// TIA Portal V19 program export: 0 tag tables, 0 data types, 1 data blocks, 22 code blocks (in call order from the OBs), 0 instance data blocks

DATA_BLOCK "DEV_7"   // DB5
{ S7_Optimized_Access := 'TRUE' }
// stored: MemoryReserve 0
   VAR
      Convoyer : "ModuleConvoyer";
   END_VAR
   VAR RETAIN
      Retains : Struct
         ConvoyerA : Struct
            ProducedUnits : DInt;
            "Type" : SInt;
         END_STRUCT;
         ConvoyerB : Struct
            ProducedUnits : DInt;
            "Type" : SInt;
         END_STRUCT;
      END_STRUCT;
      Recipes : Struct
         Convoyer : Struct
            "A" : Struct
               "Type" : SInt;
               StampingPL : Struct
                  Enable : Bool := TRUE;
                  Double : Bool;
                  SecondPush : Bool;
                  SecondPreasure : Real;
                  RegularPreasure : Real := 1.3;
                  MaxPreasure : Real := 4.0;
                  TimerMaxPreasure : Time := T#1300ms;
                  TimerStamping : Time := T#400ms;
                  TimerSecond : Time;
               END_STRUCT;
               SettingsPL : Struct
                  Camera : Bool := TRUE;
                  Blow : Bool := TRUE;
                  BlowTime : Time := T#1000ms;
               END_STRUCT;
               StampingCN : Struct
                  Enable : Bool := TRUE;
                  Double : Bool;
                  SecondPush : Bool := TRUE;
                  SecondPreasure : Real := 4.0;
                  RegularPreasure : Real := 1.3;
                  MaxPreasure : Real := 4.5;
                  TimerMaxPreasure : Time := T#1300ms;
                  TimerStamping : Time := T#800ms;
                  TimerSecond : Time := T#500ms;
               END_STRUCT;
               SettingsCN : Struct
                  Camera : Bool := TRUE;
                  Blow : Bool := TRUE;
                  BlowTime : Time := T#1000ms;
               END_STRUCT;
               StampingPlastic : Struct
                  Enable : Bool := TRUE;
                  Double : Bool;
                  SecondPush : Bool;
                  SecondPreasure : Real;
                  RegularPreasure : Real := 1.3;
                  MaxPreasure : Real := 4.0;
                  TimerMaxPreasure : Time := T#1300ms;
                  TimerStamping : Time := T#400ms;
                  TimerSecond : Time;
               END_STRUCT;
               SettingsPlastic : Struct
                  Camera : Bool := TRUE;
                  Blow : Bool := TRUE;
                  BlowTime : Time := T#1000ms;
               END_STRUCT;
               StampingTransport : Struct
                  Enable : Bool := FALSE;
                  Double : Bool := FALSE;
                  SecondPush : Bool := FALSE;
                  SecondPreasure : Real;
                  RegularPreasure : Real := 1.3;
                  MaxPreasure : Real := 4.0;
                  TimerMaxPreasure : Time := T#1300ms;
                  TimerStamping : Time := T#400ms;
                  TimerSecond : Time;
               END_STRUCT;
               SettingsTransport : Struct
                  Camera : Bool := FALSE;
                  Blow : Bool := FALSE;
                  BlowTime : Time := T#1000ms;
               END_STRUCT;
            END_STRUCT;
            "B" : Struct
               "Type" : SInt;
               StampingPL : Struct
                  Enable : Bool := TRUE;
                  Double : Bool;
                  SecondPush : Bool;
                  SecondPreasure : Real;
                  RegularPreasure : Real := 1.3;
                  MaxPreasure : Real := 4.0;
                  TimerMaxPreasure : Time := T#1300ms;
                  TimerStamping : Time := T#400ms;
                  TimerSecond : Time;
               END_STRUCT;
               SettingsPL : Struct
                  Camera : Bool := TRUE;
                  Blow : Bool := TRUE;
                  BlowTime : Time := T#1000ms;
               END_STRUCT;
               StampingCN : Struct
                  Enable : Bool := TRUE;
                  Double : Bool;
                  SecondPush : Bool := TRUE;
                  SecondPreasure : Real := 4.0;
                  RegularPreasure : Real := 1.3;
                  MaxPreasure : Real := 4.5;
                  TimerMaxPreasure : Time := T#1300ms;
                  TimerStamping : Time := T#800ms;
                  TimerSecond : Time := T#500ms;
               END_STRUCT;
               SettingsCN : Struct
                  Camera : Bool := TRUE;
                  Blow : Bool := TRUE;
                  BlowTime : Time := T#1000ms;
               END_STRUCT;
               StampingPlastic : Struct
                  Enable : Bool := TRUE;
                  Double : Bool;
                  SecondPush : Bool;
                  SecondPreasure : Real;
                  RegularPreasure : Real := 1.3;
                  MaxPreasure : Real := 4.0;
                  TimerMaxPreasure : Time := T#1300ms;
                  TimerStamping : Time := T#400ms;
                  TimerSecond : Time;
               END_STRUCT;
               SettingsPlastic : Struct
                  Camera : Bool := TRUE;
                  Blow : Bool := TRUE;
                  BlowTime : Time := T#1000ms;
               END_STRUCT;
               StampingTransport : Struct
                  Enable : Bool := FALSE;
                  Double : Bool := FALSE;
                  SecondPush : Bool := FALSE;
                  SecondPreasure : Real;
                  RegularPreasure : Real := 1.3;
                  MaxPreasure : Real := 4.0;
                  TimerMaxPreasure : Time := T#1300ms;
                  TimerStamping : Time := T#400ms;
                  TimerSecond : Time;
               END_STRUCT;
               SettingsTransport : Struct
                  Camera : Bool := FALSE;
                  Blow : Bool := FALSE;
                  BlowTime : Time := T#1000ms;
               END_STRUCT;
            END_STRUCT;
         END_STRUCT;
      END_STRUCT;
      OPC : Struct
         Convoyer : Struct
            "A" : Struct
               LifetimeProduction : DInt;
               CycleTime : Time;
               CameraCycle : Time;
               StampingCycle : Time;
               ActualRecipe : WString[30];
               Status : Struct
                  ReadyToWork : Bool;
                  Working : Bool;
                  Error : Bool;
               END_STRUCT;
            END_STRUCT;
            "B" : Struct
               LifetimeProduction : DInt;
               CycleTime : Time;
               CameraCycle : Time;
               StampingCycle : Time;
               ActualRecipe : WString[30];
               Status : Struct
                  ReadyToWork : Bool;
                  Working : Bool;
                  Error : Bool;
               END_STRUCT;
            END_STRUCT;
         END_STRUCT;
      END_STRUCT;
   END_VAR
BEGIN
   Convoyer.Modular_A.CameraConnection.InterfaceId := 64;
   Convoyer.Modular_A.CameraConnection.ID := 1;
   Convoyer.Modular_A.CameraConnection.ConnectionType := 16#0B;
   Convoyer.Modular_A.CameraConnection.ActiveEstablished := false;
   Convoyer.Modular_A.CameraConnection.RemoteAddress.ADDR[1] := 192;
   Convoyer.Modular_A.CameraConnection.RemoteAddress.ADDR[2] := 168;
   Convoyer.Modular_A.CameraConnection.RemoteAddress.ADDR[3] := 0;
   Convoyer.Modular_A.CameraConnection.RemoteAddress.ADDR[4] := 70;
   Convoyer.Modular_A.CameraConnection.RemotePort := 0;
   Convoyer.Modular_A.CameraConnection.LocalPort := 2137;
   Convoyer.Modular_A.Pneumatics.Stamping.Timers.In := T#6000ms;
   Convoyer.Modular_A.Pneumatics.Stamping.Timers.Out := T#5000ms;
   Convoyer.Modular_A.Pneumatics.IVT.Sensor.Analog.SetValue := 0.0;
   Convoyer.Modular_A.Pneumatics.IVT.Sensor.Settings.Min := 0.0;
   Convoyer.Modular_A.Pneumatics.IVT.Sensor.Settings.Max := 7.0;
   Convoyer.Modular_A.HMI.Camera.Enable := TRUE;
   Convoyer.Modular_A.HMI.Camera.TimerConnection := T#100000ms;
   Convoyer.Modular_A.HMI.Stamping.Enable := TRUE;
   Convoyer.Modular_A.HMI.Stamping.RegularPreasure := 3.0;
   Convoyer.Modular_A.HMI.Stamping.MaxPreasure := 6.0;
   Convoyer.Modular_A.HMI.Stamping.TimerMaxPreasure := T#1500ms;
   Convoyer.Modular_A.HMI.Stamping.TimerStamping := T#1000ms;
   Convoyer.Modular_A.HMI.Blow.Enable := TRUE;
   Convoyer.Modular_A.HMI.Blow."Time" := T#1000ms;
   Convoyer.Modular_B.CameraConnection.InterfaceId := 64;
   Convoyer.Modular_B.CameraConnection.ID := 16#2;
   Convoyer.Modular_B.CameraConnection.ConnectionType := 16#0B;
   Convoyer.Modular_B.CameraConnection.ActiveEstablished := FALSE;
   Convoyer.Modular_B.CameraConnection.RemoteAddress.ADDR[1] := 192;
   Convoyer.Modular_B.CameraConnection.RemoteAddress.ADDR[2] := 168;
   Convoyer.Modular_B.CameraConnection.RemoteAddress.ADDR[3] := 0;
   Convoyer.Modular_B.CameraConnection.RemoteAddress.ADDR[4] := 71;
   Convoyer.Modular_B.CameraConnection.RemotePort := 0;
   Convoyer.Modular_B.CameraConnection.LocalPort := 2137;
END_DATA_BLOCK

ORGANIZATION_BLOCK "Main"   // OB1, LAD, ProgramCycle
TITLE = "Main Program Sweep (Cycle)"
{ S7_Optimized_Access := 'TRUE' }
// stored: SetENOAutomatically false
   VAR_INPUT
      Initial_Call : Bool;   // Initial call of this OB
      Remanence : Bool;   // =True, if remanent data are available
   END_VAR
BEGIN

REGION Network 1
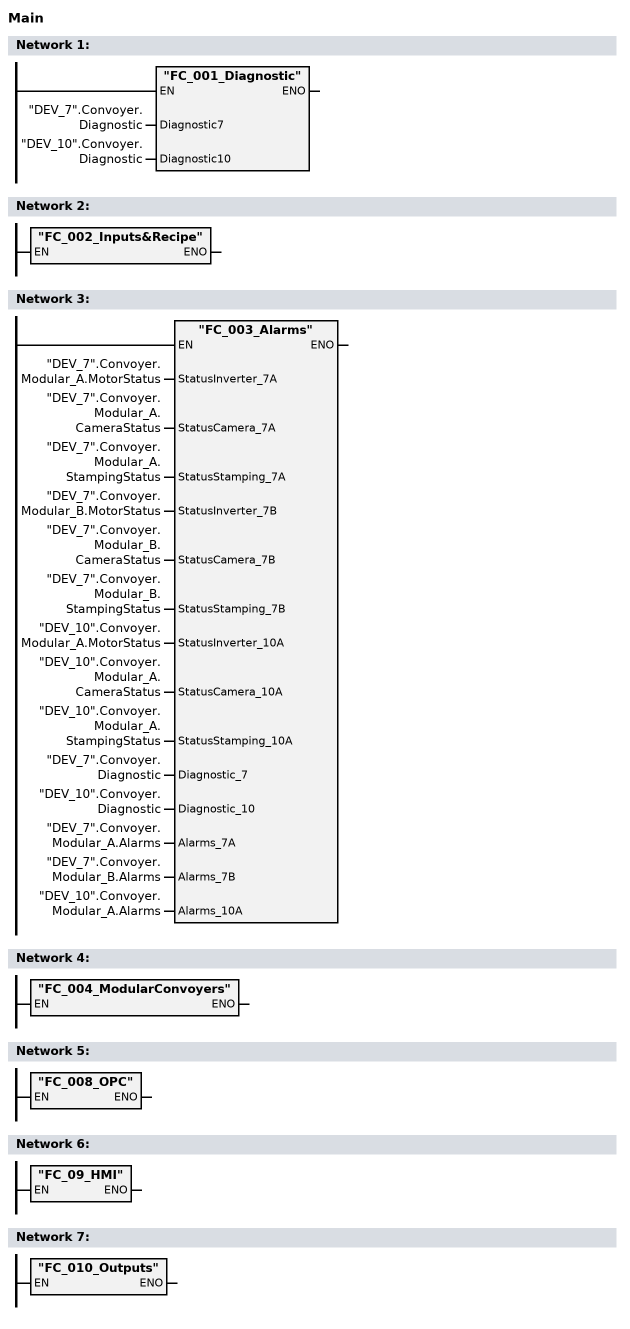
   RUNG wire#powerrail
      "FC_001_Diagnostic"(Diagnostic7 := "DEV_7".Convoyer.Diagnostic, Diagnostic10 := "DEV_10".Convoyer.Diagnostic)
   END_RUNG
   // the same network as SCL:
   "FC_001_Diagnostic"(Diagnostic7 := "DEV_7".Convoyer.Diagnostic, Diagnostic10 := "DEV_10".Convoyer.Diagnostic);
END_REGION

REGION Network 2
   RUNG wire#powerrail
      "FC_002_Inputs&Recipe"()
   END_RUNG
   // the same network as SCL:
   "FC_002_Inputs&Recipe"();
END_REGION

REGION Network 3
   RUNG wire#powerrail
      "FC_003_Alarms"(StatusInverter_7A := "DEV_7".Convoyer.Modular_A.MotorStatus, StatusCamera_7A := "DEV_7".Convoyer.Modular_A.CameraStatus, StatusStamping_7A := "DEV_7".Convoyer.Modular_A.StampingStatus, StatusInverter_7B := "DEV_7".Convoyer.Modular_B.MotorStatus, StatusCamera_7B := "DEV_7".Convoyer.Modular_B.CameraStatus, StatusStamping_7B := "DEV_7".Convoyer.Modular_B.StampingStatus, StatusInverter_10A := "DEV_10".Convoyer.Modular_A.MotorStatus, StatusCamera_10A := "DEV_10".Convoyer.Modular_A.CameraStatus, StatusStamping_10A := "DEV_10".Convoyer.Modular_A.StampingStatus, Diagnostic_7 := "DEV_7".Convoyer.Diagnostic, Diagnostic_10 := "DEV_10".Convoyer.Diagnostic, Alarms_7A := "DEV_7".Convoyer.Modular_A.Alarms, Alarms_7B := "DEV_7".Convoyer.Modular_B.Alarms, Alarms_10A := "DEV_10".Convoyer.Modular_A.Alarms)
   END_RUNG
   // the same network as SCL:
   "FC_003_Alarms"(StatusInverter_7A := "DEV_7".Convoyer.Modular_A.MotorStatus,
                   StatusCamera_7A := "DEV_7".Convoyer.Modular_A.CameraStatus,
                   StatusStamping_7A := "DEV_7".Convoyer.Modular_A.StampingStatus,
                   StatusInverter_7B := "DEV_7".Convoyer.Modular_B.MotorStatus,
                   StatusCamera_7B := "DEV_7".Convoyer.Modular_B.CameraStatus,
                   StatusStamping_7B := "DEV_7".Convoyer.Modular_B.StampingStatus,
                   StatusInverter_10A := "DEV_10".Convoyer.Modular_A.MotorStatus,
                   StatusCamera_10A := "DEV_10".Convoyer.Modular_A.CameraStatus,
                   StatusStamping_10A := "DEV_10".Convoyer.Modular_A.StampingStatus,
                   Diagnostic_7 := "DEV_7".Convoyer.Diagnostic,
                   Diagnostic_10 := "DEV_10".Convoyer.Diagnostic,
                   Alarms_7A := "DEV_7".Convoyer.Modular_A.Alarms,
                   Alarms_7B := "DEV_7".Convoyer.Modular_B.Alarms,
                   Alarms_10A := "DEV_10".Convoyer.Modular_A.Alarms);
END_REGION

REGION Network 4
   RUNG wire#powerrail
      "FC_004_ModularConvoyers"()
   END_RUNG
   // the same network as SCL:
   "FC_004_ModularConvoyers"();
END_REGION

REGION Network 5
   RUNG wire#powerrail
      "FC_008_OPC"()
   END_RUNG
   // the same network as SCL:
   "FC_008_OPC"();
END_REGION

REGION Network 6
   RUNG wire#powerrail
      "FC_09_HMI"()
   END_RUNG
   // the same network as SCL:
   "FC_09_HMI"();
END_REGION

REGION Network 7
   RUNG wire#powerrail
      "FC_010_Outputs"()
   END_RUNG
   // the same network as SCL:
   "FC_010_Outputs"();
END_REGION
END_ORGANIZATION_BLOCK

FUNCTION "FC_001_Diagnostic" : Void   // FC12, LAD
{ S7_Optimized_Access := 'TRUE' }
// stored: SetENOAutomatically false
   VAR_IN_OUT
      Diagnostic7 : "DiagnosticMainCabinet";
      Diagnostic10 : "DiagnosticMainCabinet";
   END_VAR
BEGIN

REGION Network 1 (SCL)
   //************************************************************
   //===Author: Mateusz Połojko
   //-----Linkedin: https://pl.linkedin.com/in/mateusz-po%C5%82ojko-52a3541b1
   //-----Github: https://github.com/Bhazel95
   //===Description:
   //-----Diagnostic of hardware components
   //===Customer:
   //-----Apator Powogaz S.A.
   //************************************************************
END_REGION

REGION Network 2 (SCL)
   //Transporter 7A & 7B
   #Diagnostic7.ET_200SP.HeadModule_0.LADDR:= "IO_device_1~Head";
   #Diagnostic7.ET_200SP.HeadModule_0.Mode := 1;

   #Diagnostic7.ET_200SP.BusAdapter_1.LADDR := "IO_device_1~BusAdapter-Send_1xFC_1";
   #Diagnostic7.ET_200SP.BusAdapter_1.Mode := 1;

   #Diagnostic7.ET_200SP.InputSafety_2.LADDR := "IO_device_1~F-DI_8x24VDC_HF_1" ;
   #Diagnostic7.ET_200SP.InputSafety_2.Mode := 1;

   #Diagnostic7.ET_200SP.InputSafety_3.LADDR := "IO_device_1~F-DI_8x24VDC_HF_2";
   #Diagnostic7.ET_200SP.InputSafety_3.Mode := 1;

   #Diagnostic7.ET_200SP.InputSafety_4.LADDR := "IO_device_1~F-DI_8x24VDC_HF_3";
   #Diagnostic7.ET_200SP.InputSafety_4.Mode := 1;

   #Diagnostic7.ET_200SP.InputSafety_5.LADDR := "IO_device_1~F-DI_8x24VDC_HF_5";
   #Diagnostic7.ET_200SP.InputSafety_5.Mode := 1;

   #Diagnostic7.ET_200SP.InputSafety_6.LADDR := "IO_device_1~F-DI_8x24VDC_HF_4";
   #Diagnostic7.ET_200SP.InputSafety_6.Mode := 1;

   #Diagnostic7.ET_200SP.OutputSafety_7.LADDR := "IO_device_1~F-DQ_8x24VDC_0_5A_PP_HF_1";
   #Diagnostic7.ET_200SP.OutputSafety_7.Mode := 1;

   #Diagnostic7.ET_200SP.RelaySafety_9.LADDR := "IO_device_1~F-RQ_1x24__48VDC_24__230VAC_5A_1";
   #Diagnostic7.ET_200SP.RelaySafety_9.Mode := 1;

   #Diagnostic7.ET_200SP.RelaySafety_10.LADDR := "IO_device_1~F-RQ_1x24__48VDC_24__230VAC_5A_2";
   #Diagnostic7.ET_200SP.RelaySafety_10.Mode := 1;

   #Diagnostic7.ET_200SP.InputsDigital_11.LADDR := "IO_device_1~DI_16x24VDC_ST_1";
   #Diagnostic7.ET_200SP.InputsDigital_11.Mode := 1;

   #Diagnostic7.ET_200SP.InputsDigital_12.LADDR := "IO_device_1~DI_16x24VDC_ST_2";
   #Diagnostic7.ET_200SP.InputsDigital_12.Mode := 1;

   #Diagnostic7.ET_200SP.InputsDigital_13.LADDR := "IO_device_1~DI_16x24VDC_ST_3";
   #Diagnostic7.ET_200SP.InputsDigital_13.Mode := 1;

   #Diagnostic7.ET_200SP.InputAnalog_14.LADDR := "IO_device_1~AI_2xI_2-_4-wire_ST_1";
   #Diagnostic7.ET_200SP.InputAnalog_14.Mode := 1;

   #Diagnostic7.ET_200SP.OutputDigital_15.LADDR := "IO_device_1~DQ_16x24VDC_0_5A_ST_1";
   #Diagnostic7.ET_200SP.OutputDigital_15.Mode := 1;

   #Diagnostic7.ET_200SP.OutputDigital_16.LADDR := "IO_device_1~DQ_16x24VDC_0_5A_ST_2";
   #Diagnostic7.ET_200SP.OutputDigital_16.Mode := 1;

   #Diagnostic7.ET_200SP.OutputDigital_17.LADDR := "IO_device_1~DQ_16x24VDC_0_5A_ST_3";
   #Diagnostic7.ET_200SP.OutputDigital_17.Mode := 1;

   #Diagnostic7.ET_200SP.OutputDigital_18.LADDR := "IO_device_1~DQ_16x24VDC_0_5A_ST_4";
   #Diagnostic7.ET_200SP.OutputDigital_18.Mode := 1;

   #Diagnostic7.ET_200SP.OutputAnalog_19.LADDR := "IO_device_1~AQ_2xI_ST_1";
   #Diagnostic7.ET_200SP.OutputAnalog_19.Mode := 1;

   #Diagnostic7.ET_200SP.ET_200AL_1.LADDR := "IO_device_1~DI_8x24VDC_8xM8_1";
   #Diagnostic7.ET_200SP.ET_200AL_1.Mode := 1;

   #Diagnostic7.ET_200SP.ET_200AL_2.LADDR := "IO_device_1~DI_8x24VDC_8xM8_2";
   #Diagnostic7.ET_200SP.ET_200AL_2.Mode := 1;


   #Diagnostic7.SinamicG120_1.LADDR := "G120_CU250S_2_PN_VECTOR_7A~PROFINET_interface~IODevice";
   #Diagnostic7.SinamicG120_1.Mode := 1;

   #Diagnostic7.SinamicG120_1.LADDR := "G120_CU250S_2_PN_VECTOR_7B~PROFINET_interface~IODevice";
   #Diagnostic7.SinamicG120_1.Mode := 1;
END_REGION

REGION Network 3 (SCL)
   //Transporter 10A & 10B
   #Diagnostic10.ET_200SP.HeadModule_0.LADDR := "IO_device_2~Head";
   #Diagnostic10.ET_200SP.HeadModule_0.Mode := 1;

   #Diagnostic10.ET_200SP.BusAdapter_1.LADDR := "IO_device_2~BusAdapter-Send_1xFC_1";
   #Diagnostic10.ET_200SP.BusAdapter_1.Mode := 1;

   #Diagnostic10.ET_200SP.InputSafety_2.LADDR := "IO_device_2~F-DI_8x24VDC_HF_1";
   #Diagnostic10.ET_200SP.InputSafety_2.Mode := 1;

   #Diagnostic10.ET_200SP.InputSafety_3.LADDR := "IO_device_2~F-DI_8x24VDC_HF_2";
   #Diagnostic10.ET_200SP.InputSafety_3.Mode := 1;

   #Diagnostic10.ET_200SP.InputSafety_4.LADDR := "IO_device_2~F-DI_8x24VDC_HF_3";
   #Diagnostic10.ET_200SP.InputSafety_4.Mode := 1;

   #Diagnostic10.ET_200SP.InputSafety_5.LADDR := "IO_device_2~F-DI_8x24VDC_HF_4";
   #Diagnostic10.ET_200SP.InputSafety_5.Mode := 1;

   #Diagnostic10.ET_200SP.InputSafety_6.LADDR := "IO_device_2~F-DI_8x24VDC_HF_5";
   #Diagnostic10.ET_200SP.InputSafety_6.Mode := 1;

   #Diagnostic10.ET_200SP.OutputSafety_7.LADDR := "IO_device_2~F-DQ_8x24VDC_0_5A_PP_HF_1";
   #Diagnostic10.ET_200SP.OutputSafety_7.Mode := 1;

   #Diagnostic10.ET_200SP.RelaySafety_9.LADDR := "IO_device_2~F-RQ_1x24__48VDC_24__230VAC_5A_1";
   #Diagnostic10.ET_200SP.RelaySafety_9.Mode := 1;

   #Diagnostic10.ET_200SP.RelaySafety_10.LADDR := "IO_device_2~F-RQ_1x24__48VDC_24__230VAC_5A_2";
   #Diagnostic10.ET_200SP.RelaySafety_10.Mode := 1;

   #Diagnostic10.ET_200SP.InputsDigital_11.LADDR := "IO_device_2~DI_16x24VDC_ST_1";
   #Diagnostic10.ET_200SP.InputsDigital_11.Mode := 1;

   #Diagnostic10.ET_200SP.InputsDigital_12.LADDR := "IO_device_2~DI_16x24VDC_ST_2";
   #Diagnostic10.ET_200SP.InputsDigital_12.Mode := 1;

   #Diagnostic10.ET_200SP.InputsDigital_13.LADDR := "IO_device_2~DI_16x24VDC_ST_3";
   #Diagnostic10.ET_200SP.InputsDigital_13.Mode := 1;

   #Diagnostic10.ET_200SP.InputAnalog_14.LADDR := "IO_device_2~AI_2xI_2-_4-wire_ST_1";
   #Diagnostic10.ET_200SP.InputAnalog_14.Mode := 1;

   #Diagnostic10.ET_200SP.OutputDigital_15.LADDR := "IO_device_2~DQ_16x24VDC_0_5A_ST_1";
   #Diagnostic10.ET_200SP.OutputDigital_15.Mode := 1;

   #Diagnostic10.ET_200SP.OutputDigital_16.LADDR := "IO_device_2~DQ_16x24VDC_0_5A_ST_2";
   #Diagnostic10.ET_200SP.OutputDigital_16.Mode := 1;

   #Diagnostic10.ET_200SP.OutputDigital_17.LADDR := "IO_device_2~DQ_16x24VDC_0_5A_ST_3";
   #Diagnostic10.ET_200SP.OutputDigital_17.Mode := 1;

   #Diagnostic10.ET_200SP.OutputDigital_18.LADDR := "IO_device_2~DQ_16x24VDC_0_5A_ST_4";
   #Diagnostic10.ET_200SP.OutputDigital_18.Mode := 1;

   #Diagnostic10.ET_200SP.OutputAnalog_19.LADDR := "IO_device_2~AQ_2xI_ST_1";
   #Diagnostic10.ET_200SP.OutputAnalog_19.Mode := 1;

   #Diagnostic10.ET_200SP.ET_200AL_1.LADDR := "IO_device_2~DI_8x24VDC_8xM8_1";
   #Diagnostic10.ET_200SP.ET_200AL_1.Mode := 1;

   #Diagnostic10.ET_200SP.ET_200AL_2.LADDR := "IO_device_2~DI_8x24VDC_8xM8_2";
   #Diagnostic10.ET_200SP.ET_200AL_2.Mode := 1;


   #Diagnostic10.SinamicG120_1.LADDR := "G120_CU250S_2_PN_VECTOR_10A~PROFINET_interface~IODevice";
   #Diagnostic10.SinamicG120_1.Mode := 1;
END_REGION

REGION Network 4
   // ET 200SP - MODUL GLOWNY 7
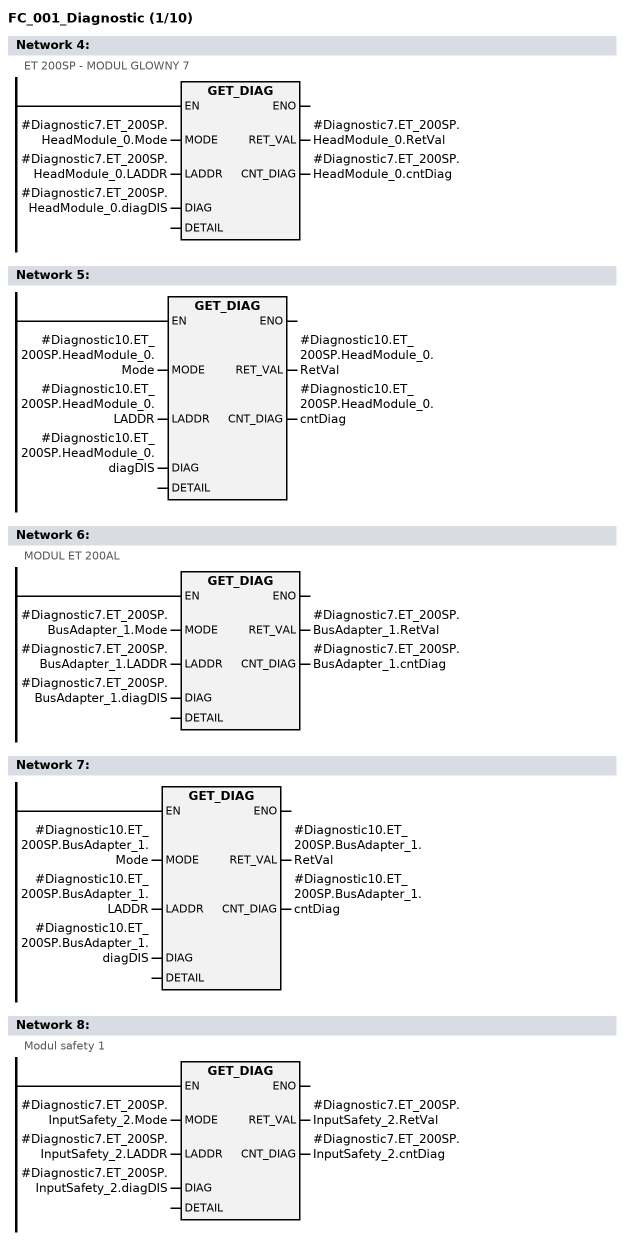
   RUNG wire#powerrail
      GET_DIAG(MODE := #Diagnostic7.ET_200SP.HeadModule_0.Mode, LADDR := #Diagnostic7.ET_200SP.HeadModule_0.LADDR, DIAG := #Diagnostic7.ET_200SP.HeadModule_0.diagDIS, DETAIL :=, RET_VAL => #Diagnostic7.ET_200SP.HeadModule_0.RetVal, CNT_DIAG => #Diagnostic7.ET_200SP.HeadModule_0.cntDiag)
   END_RUNG
   // the same network as SCL:
   #Diagnostic7.ET_200SP.HeadModule_0.RetVal := GET_DIAG(MODE := #Diagnostic7.ET_200SP.HeadModule_0.Mode,
                           LADDR := #Diagnostic7.ET_200SP.HeadModule_0.LADDR,
                           DIAG := #Diagnostic7.ET_200SP.HeadModule_0.diagDIS,
                           CNT_DIAG => #Diagnostic7.ET_200SP.HeadModule_0.cntDiag);
END_REGION

REGION Network 5
   RUNG wire#powerrail
      GET_DIAG(MODE := #Diagnostic10.ET_200SP.HeadModule_0.Mode, LADDR := #Diagnostic10.ET_200SP.HeadModule_0.LADDR, DIAG := #Diagnostic10.ET_200SP.HeadModule_0.diagDIS, DETAIL :=, RET_VAL => #Diagnostic10.ET_200SP.HeadModule_0.RetVal, CNT_DIAG => #Diagnostic10.ET_200SP.HeadModule_0.cntDiag)
   END_RUNG
   // the same network as SCL:
   #Diagnostic10.ET_200SP.HeadModule_0.RetVal := GET_DIAG(MODE := #Diagnostic10.ET_200SP.HeadModule_0.Mode,
                           LADDR := #Diagnostic10.ET_200SP.HeadModule_0.LADDR,
                           DIAG := #Diagnostic10.ET_200SP.HeadModule_0.diagDIS,
                           CNT_DIAG => #Diagnostic10.ET_200SP.HeadModule_0.cntDiag);
END_REGION

REGION Network 6
   // MODUL ET 200AL
   RUNG wire#powerrail
      GET_DIAG(MODE := #Diagnostic7.ET_200SP.BusAdapter_1.Mode, LADDR := #Diagnostic7.ET_200SP.BusAdapter_1.LADDR, DIAG := #Diagnostic7.ET_200SP.BusAdapter_1.diagDIS, DETAIL :=, RET_VAL => #Diagnostic7.ET_200SP.BusAdapter_1.RetVal, CNT_DIAG => #Diagnostic7.ET_200SP.BusAdapter_1.cntDiag)
   END_RUNG
   // the same network as SCL:
   #Diagnostic7.ET_200SP.BusAdapter_1.RetVal := GET_DIAG(MODE := #Diagnostic7.ET_200SP.BusAdapter_1.Mode,
                           LADDR := #Diagnostic7.ET_200SP.BusAdapter_1.LADDR,
                           DIAG := #Diagnostic7.ET_200SP.BusAdapter_1.diagDIS,
                           CNT_DIAG => #Diagnostic7.ET_200SP.BusAdapter_1.cntDiag);
END_REGION

REGION Network 7
   RUNG wire#powerrail
      GET_DIAG(MODE := #Diagnostic10.ET_200SP.BusAdapter_1.Mode, LADDR := #Diagnostic10.ET_200SP.BusAdapter_1.LADDR, DIAG := #Diagnostic10.ET_200SP.BusAdapter_1.diagDIS, DETAIL :=, RET_VAL => #Diagnostic10.ET_200SP.BusAdapter_1.RetVal, CNT_DIAG => #Diagnostic10.ET_200SP.BusAdapter_1.cntDiag)
   END_RUNG
   // the same network as SCL:
   #Diagnostic10.ET_200SP.BusAdapter_1.RetVal := GET_DIAG(MODE := #Diagnostic10.ET_200SP.BusAdapter_1.Mode,
                           LADDR := #Diagnostic10.ET_200SP.BusAdapter_1.LADDR,
                           DIAG := #Diagnostic10.ET_200SP.BusAdapter_1.diagDIS,
                           CNT_DIAG => #Diagnostic10.ET_200SP.BusAdapter_1.cntDiag);
END_REGION

REGION Network 8
   // Modul safety 1
   RUNG wire#powerrail
      GET_DIAG(MODE := #Diagnostic7.ET_200SP.InputSafety_2.Mode, LADDR := #Diagnostic7.ET_200SP.InputSafety_2.LADDR, DIAG := #Diagnostic7.ET_200SP.InputSafety_2.diagDIS, DETAIL :=, RET_VAL => #Diagnostic7.ET_200SP.InputSafety_2.RetVal, CNT_DIAG => #Diagnostic7.ET_200SP.InputSafety_2.cntDiag)
   END_RUNG
   // the same network as SCL:
   #Diagnostic7.ET_200SP.InputSafety_2.RetVal := GET_DIAG(MODE := #Diagnostic7.ET_200SP.InputSafety_2.Mode,
                           LADDR := #Diagnostic7.ET_200SP.InputSafety_2.LADDR,
                           DIAG := #Diagnostic7.ET_200SP.InputSafety_2.diagDIS,
                           CNT_DIAG => #Diagnostic7.ET_200SP.InputSafety_2.cntDiag);
END_REGION

REGION Network 9
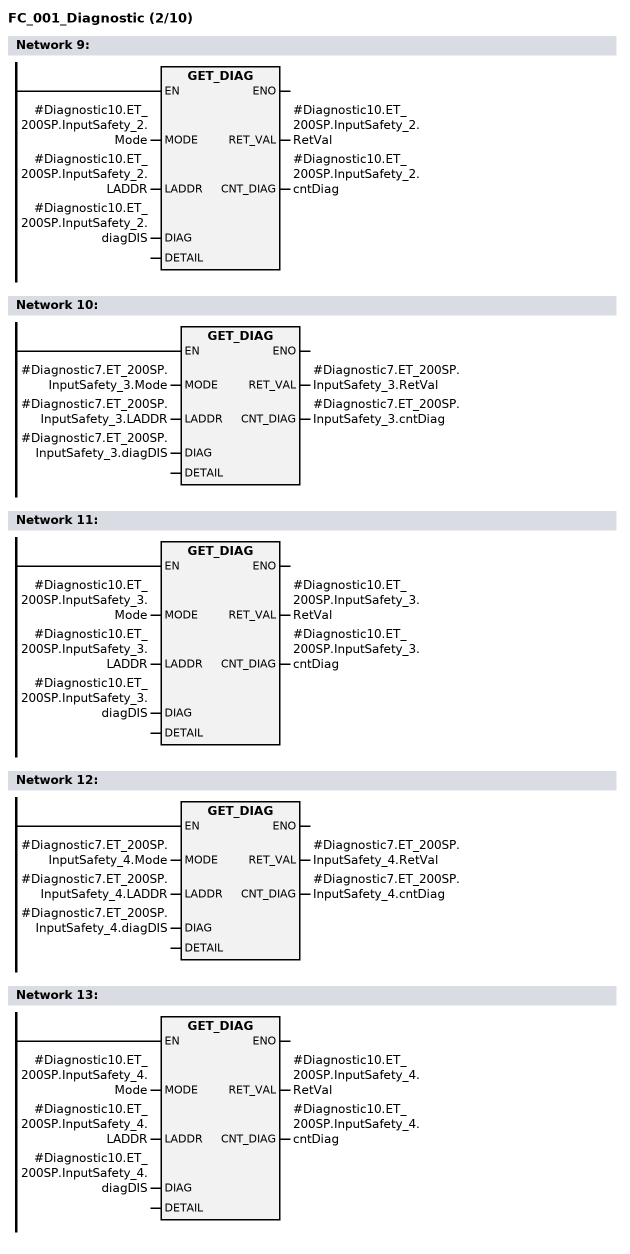
   RUNG wire#powerrail
      GET_DIAG(MODE := #Diagnostic10.ET_200SP.InputSafety_2.Mode, LADDR := #Diagnostic10.ET_200SP.InputSafety_2.LADDR, DIAG := #Diagnostic10.ET_200SP.InputSafety_2.diagDIS, DETAIL :=, RET_VAL => #Diagnostic10.ET_200SP.InputSafety_2.RetVal, CNT_DIAG => #Diagnostic10.ET_200SP.InputSafety_2.cntDiag)
   END_RUNG
   // the same network as SCL:
   #Diagnostic10.ET_200SP.InputSafety_2.RetVal := GET_DIAG(MODE := #Diagnostic10.ET_200SP.InputSafety_2.Mode,
                           LADDR := #Diagnostic10.ET_200SP.InputSafety_2.LADDR,
                           DIAG := #Diagnostic10.ET_200SP.InputSafety_2.diagDIS,
                           CNT_DIAG => #Diagnostic10.ET_200SP.InputSafety_2.cntDiag);
END_REGION

REGION Network 10
   RUNG wire#powerrail
      GET_DIAG(MODE := #Diagnostic7.ET_200SP.InputSafety_3.Mode, LADDR := #Diagnostic7.ET_200SP.InputSafety_3.LADDR, DIAG := #Diagnostic7.ET_200SP.InputSafety_3.diagDIS, DETAIL :=, RET_VAL => #Diagnostic7.ET_200SP.InputSafety_3.RetVal, CNT_DIAG => #Diagnostic7.ET_200SP.InputSafety_3.cntDiag)
   END_RUNG
   // the same network as SCL:
   #Diagnostic7.ET_200SP.InputSafety_3.RetVal := GET_DIAG(MODE := #Diagnostic7.ET_200SP.InputSafety_3.Mode,
                           LADDR := #Diagnostic7.ET_200SP.InputSafety_3.LADDR,
                           DIAG := #Diagnostic7.ET_200SP.InputSafety_3.diagDIS,
                           CNT_DIAG => #Diagnostic7.ET_200SP.InputSafety_3.cntDiag);
END_REGION

REGION Network 11
   RUNG wire#powerrail
      GET_DIAG(MODE := #Diagnostic10.ET_200SP.InputSafety_3.Mode, LADDR := #Diagnostic10.ET_200SP.InputSafety_3.LADDR, DIAG := #Diagnostic10.ET_200SP.InputSafety_3.diagDIS, DETAIL :=, RET_VAL => #Diagnostic10.ET_200SP.InputSafety_3.RetVal, CNT_DIAG => #Diagnostic10.ET_200SP.InputSafety_3.cntDiag)
   END_RUNG
   // the same network as SCL:
   #Diagnostic10.ET_200SP.InputSafety_3.RetVal := GET_DIAG(MODE := #Diagnostic10.ET_200SP.InputSafety_3.Mode,
                           LADDR := #Diagnostic10.ET_200SP.InputSafety_3.LADDR,
                           DIAG := #Diagnostic10.ET_200SP.InputSafety_3.diagDIS,
                           CNT_DIAG => #Diagnostic10.ET_200SP.InputSafety_3.cntDiag);
END_REGION

REGION Network 12
   RUNG wire#powerrail
      GET_DIAG(MODE := #Diagnostic7.ET_200SP.InputSafety_4.Mode, LADDR := #Diagnostic7.ET_200SP.InputSafety_4.LADDR, DIAG := #Diagnostic7.ET_200SP.InputSafety_4.diagDIS, DETAIL :=, RET_VAL => #Diagnostic7.ET_200SP.InputSafety_4.RetVal, CNT_DIAG => #Diagnostic7.ET_200SP.InputSafety_4.cntDiag)
   END_RUNG
   // the same network as SCL:
   #Diagnostic7.ET_200SP.InputSafety_4.RetVal := GET_DIAG(MODE := #Diagnostic7.ET_200SP.InputSafety_4.Mode,
                           LADDR := #Diagnostic7.ET_200SP.InputSafety_4.LADDR,
                           DIAG := #Diagnostic7.ET_200SP.InputSafety_4.diagDIS,
                           CNT_DIAG => #Diagnostic7.ET_200SP.InputSafety_4.cntDiag);
END_REGION

REGION Network 13
   RUNG wire#powerrail
      GET_DIAG(MODE := #Diagnostic10.ET_200SP.InputSafety_4.Mode, LADDR := #Diagnostic10.ET_200SP.InputSafety_4.LADDR, DIAG := #Diagnostic10.ET_200SP.InputSafety_4.diagDIS, DETAIL :=, RET_VAL => #Diagnostic10.ET_200SP.InputSafety_4.RetVal, CNT_DIAG => #Diagnostic10.ET_200SP.InputSafety_4.cntDiag)
   END_RUNG
   // the same network as SCL:
   #Diagnostic10.ET_200SP.InputSafety_4.RetVal := GET_DIAG(MODE := #Diagnostic10.ET_200SP.InputSafety_4.Mode,
                           LADDR := #Diagnostic10.ET_200SP.InputSafety_4.LADDR,
                           DIAG := #Diagnostic10.ET_200SP.InputSafety_4.diagDIS,
                           CNT_DIAG => #Diagnostic10.ET_200SP.InputSafety_4.cntDiag);
END_REGION

REGION Network 14
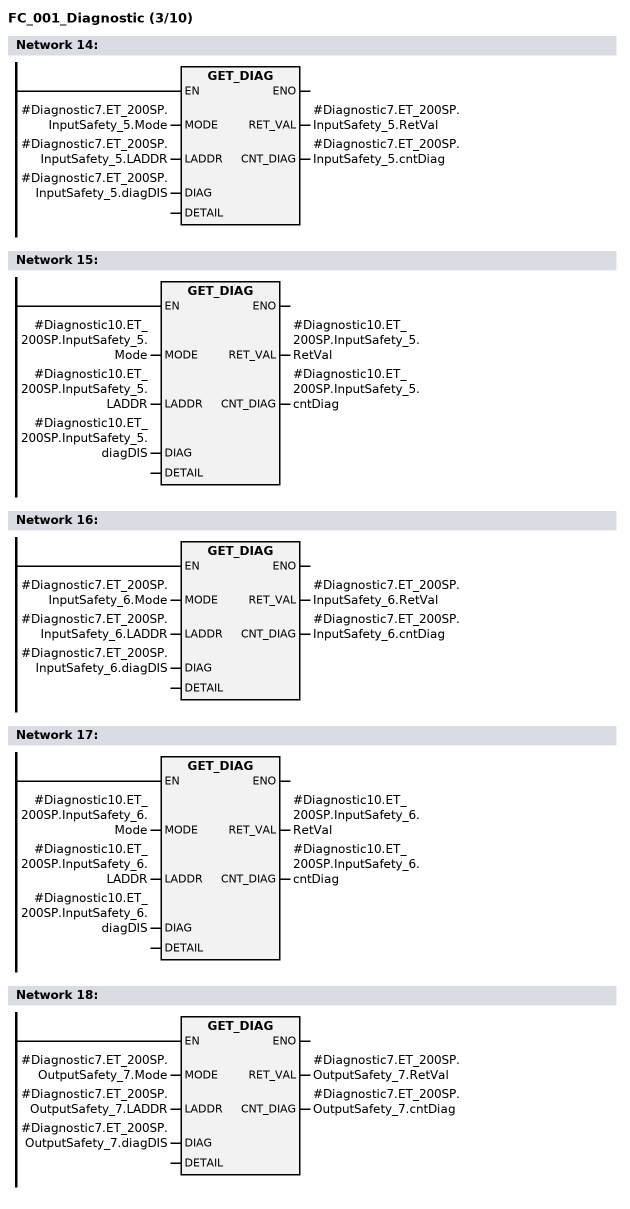
   RUNG wire#powerrail
      GET_DIAG(MODE := #Diagnostic7.ET_200SP.InputSafety_5.Mode, LADDR := #Diagnostic7.ET_200SP.InputSafety_5.LADDR, DIAG := #Diagnostic7.ET_200SP.InputSafety_5.diagDIS, DETAIL :=, RET_VAL => #Diagnostic7.ET_200SP.InputSafety_5.RetVal, CNT_DIAG => #Diagnostic7.ET_200SP.InputSafety_5.cntDiag)
   END_RUNG
   // the same network as SCL:
   #Diagnostic7.ET_200SP.InputSafety_5.RetVal := GET_DIAG(MODE := #Diagnostic7.ET_200SP.InputSafety_5.Mode,
                           LADDR := #Diagnostic7.ET_200SP.InputSafety_5.LADDR,
                           DIAG := #Diagnostic7.ET_200SP.InputSafety_5.diagDIS,
                           CNT_DIAG => #Diagnostic7.ET_200SP.InputSafety_5.cntDiag);
END_REGION

REGION Network 15
   RUNG wire#powerrail
      GET_DIAG(MODE := #Diagnostic10.ET_200SP.InputSafety_5.Mode, LADDR := #Diagnostic10.ET_200SP.InputSafety_5.LADDR, DIAG := #Diagnostic10.ET_200SP.InputSafety_5.diagDIS, DETAIL :=, RET_VAL => #Diagnostic10.ET_200SP.InputSafety_5.RetVal, CNT_DIAG => #Diagnostic10.ET_200SP.InputSafety_5.cntDiag)
   END_RUNG
   // the same network as SCL:
   #Diagnostic10.ET_200SP.InputSafety_5.RetVal := GET_DIAG(MODE := #Diagnostic10.ET_200SP.InputSafety_5.Mode,
                           LADDR := #Diagnostic10.ET_200SP.InputSafety_5.LADDR,
                           DIAG := #Diagnostic10.ET_200SP.InputSafety_5.diagDIS,
                           CNT_DIAG => #Diagnostic10.ET_200SP.InputSafety_5.cntDiag);
END_REGION

REGION Network 16
   RUNG wire#powerrail
      GET_DIAG(MODE := #Diagnostic7.ET_200SP.InputSafety_6.Mode, LADDR := #Diagnostic7.ET_200SP.InputSafety_6.LADDR, DIAG := #Diagnostic7.ET_200SP.InputSafety_6.diagDIS, DETAIL :=, RET_VAL => #Diagnostic7.ET_200SP.InputSafety_6.RetVal, CNT_DIAG => #Diagnostic7.ET_200SP.InputSafety_6.cntDiag)
   END_RUNG
   // the same network as SCL:
   #Diagnostic7.ET_200SP.InputSafety_6.RetVal := GET_DIAG(MODE := #Diagnostic7.ET_200SP.InputSafety_6.Mode,
                           LADDR := #Diagnostic7.ET_200SP.InputSafety_6.LADDR,
                           DIAG := #Diagnostic7.ET_200SP.InputSafety_6.diagDIS,
                           CNT_DIAG => #Diagnostic7.ET_200SP.InputSafety_6.cntDiag);
END_REGION

REGION Network 17
   RUNG wire#powerrail
      GET_DIAG(MODE := #Diagnostic10.ET_200SP.InputSafety_6.Mode, LADDR := #Diagnostic10.ET_200SP.InputSafety_6.LADDR, DIAG := #Diagnostic10.ET_200SP.InputSafety_6.diagDIS, DETAIL :=, RET_VAL => #Diagnostic10.ET_200SP.InputSafety_6.RetVal, CNT_DIAG => #Diagnostic10.ET_200SP.InputSafety_6.cntDiag)
   END_RUNG
   // the same network as SCL:
   #Diagnostic10.ET_200SP.InputSafety_6.RetVal := GET_DIAG(MODE := #Diagnostic10.ET_200SP.InputSafety_6.Mode,
                           LADDR := #Diagnostic10.ET_200SP.InputSafety_6.LADDR,
                           DIAG := #Diagnostic10.ET_200SP.InputSafety_6.diagDIS,
                           CNT_DIAG => #Diagnostic10.ET_200SP.InputSafety_6.cntDiag);
END_REGION

REGION Network 18
   RUNG wire#powerrail
      GET_DIAG(MODE := #Diagnostic7.ET_200SP.OutputSafety_7.Mode, LADDR := #Diagnostic7.ET_200SP.OutputSafety_7.LADDR, DIAG := #Diagnostic7.ET_200SP.OutputSafety_7.diagDIS, DETAIL :=, RET_VAL => #Diagnostic7.ET_200SP.OutputSafety_7.RetVal, CNT_DIAG => #Diagnostic7.ET_200SP.OutputSafety_7.cntDiag)
   END_RUNG
   // the same network as SCL:
   #Diagnostic7.ET_200SP.OutputSafety_7.RetVal := GET_DIAG(MODE := #Diagnostic7.ET_200SP.OutputSafety_7.Mode,
                           LADDR := #Diagnostic7.ET_200SP.OutputSafety_7.LADDR,
                           DIAG := #Diagnostic7.ET_200SP.OutputSafety_7.diagDIS,
                           CNT_DIAG => #Diagnostic7.ET_200SP.OutputSafety_7.cntDiag);
END_REGION

REGION Network 19
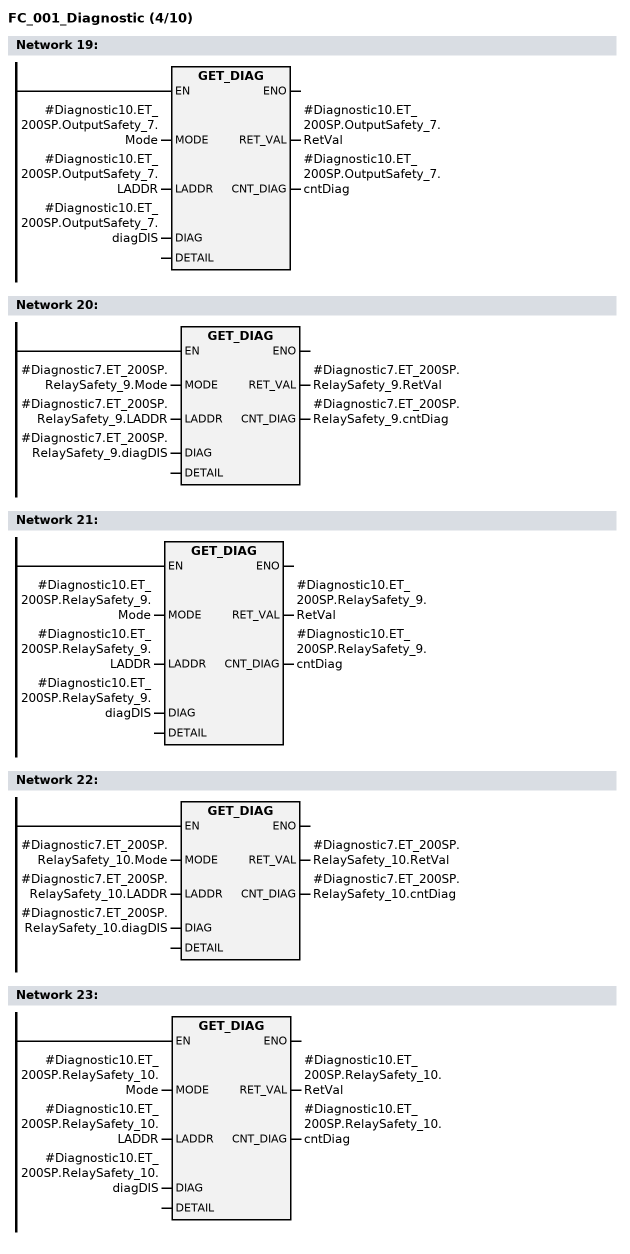
   RUNG wire#powerrail
      GET_DIAG(MODE := #Diagnostic10.ET_200SP.OutputSafety_7.Mode, LADDR := #Diagnostic10.ET_200SP.OutputSafety_7.LADDR, DIAG := #Diagnostic10.ET_200SP.OutputSafety_7.diagDIS, DETAIL :=, RET_VAL => #Diagnostic10.ET_200SP.OutputSafety_7.RetVal, CNT_DIAG => #Diagnostic10.ET_200SP.OutputSafety_7.cntDiag)
   END_RUNG
   // the same network as SCL:
   #Diagnostic10.ET_200SP.OutputSafety_7.RetVal := GET_DIAG(MODE := #Diagnostic10.ET_200SP.OutputSafety_7.Mode,
                           LADDR := #Diagnostic10.ET_200SP.OutputSafety_7.LADDR,
                           DIAG := #Diagnostic10.ET_200SP.OutputSafety_7.diagDIS,
                           CNT_DIAG => #Diagnostic10.ET_200SP.OutputSafety_7.cntDiag);
END_REGION

REGION Network 20
   RUNG wire#powerrail
      GET_DIAG(MODE := #Diagnostic7.ET_200SP.RelaySafety_9.Mode, LADDR := #Diagnostic7.ET_200SP.RelaySafety_9.LADDR, DIAG := #Diagnostic7.ET_200SP.RelaySafety_9.diagDIS, DETAIL :=, RET_VAL => #Diagnostic7.ET_200SP.RelaySafety_9.RetVal, CNT_DIAG => #Diagnostic7.ET_200SP.RelaySafety_9.cntDiag)
   END_RUNG
   // the same network as SCL:
   #Diagnostic7.ET_200SP.RelaySafety_9.RetVal := GET_DIAG(MODE := #Diagnostic7.ET_200SP.RelaySafety_9.Mode,
                           LADDR := #Diagnostic7.ET_200SP.RelaySafety_9.LADDR,
                           DIAG := #Diagnostic7.ET_200SP.RelaySafety_9.diagDIS,
                           CNT_DIAG => #Diagnostic7.ET_200SP.RelaySafety_9.cntDiag);
END_REGION

REGION Network 21
   RUNG wire#powerrail
      GET_DIAG(MODE := #Diagnostic10.ET_200SP.RelaySafety_9.Mode, LADDR := #Diagnostic10.ET_200SP.RelaySafety_9.LADDR, DIAG := #Diagnostic10.ET_200SP.RelaySafety_9.diagDIS, DETAIL :=, RET_VAL => #Diagnostic10.ET_200SP.RelaySafety_9.RetVal, CNT_DIAG => #Diagnostic10.ET_200SP.RelaySafety_9.cntDiag)
   END_RUNG
   // the same network as SCL:
   #Diagnostic10.ET_200SP.RelaySafety_9.RetVal := GET_DIAG(MODE := #Diagnostic10.ET_200SP.RelaySafety_9.Mode,
                           LADDR := #Diagnostic10.ET_200SP.RelaySafety_9.LADDR,
                           DIAG := #Diagnostic10.ET_200SP.RelaySafety_9.diagDIS,
                           CNT_DIAG => #Diagnostic10.ET_200SP.RelaySafety_9.cntDiag);
END_REGION

REGION Network 22
   RUNG wire#powerrail
      GET_DIAG(MODE := #Diagnostic7.ET_200SP.RelaySafety_10.Mode, LADDR := #Diagnostic7.ET_200SP.RelaySafety_10.LADDR, DIAG := #Diagnostic7.ET_200SP.RelaySafety_10.diagDIS, DETAIL :=, RET_VAL => #Diagnostic7.ET_200SP.RelaySafety_10.RetVal, CNT_DIAG => #Diagnostic7.ET_200SP.RelaySafety_10.cntDiag)
   END_RUNG
   // the same network as SCL:
   #Diagnostic7.ET_200SP.RelaySafety_10.RetVal := GET_DIAG(MODE := #Diagnostic7.ET_200SP.RelaySafety_10.Mode,
                           LADDR := #Diagnostic7.ET_200SP.RelaySafety_10.LADDR,
                           DIAG := #Diagnostic7.ET_200SP.RelaySafety_10.diagDIS,
                           CNT_DIAG => #Diagnostic7.ET_200SP.RelaySafety_10.cntDiag);
END_REGION

REGION Network 23
   RUNG wire#powerrail
      GET_DIAG(MODE := #Diagnostic10.ET_200SP.RelaySafety_10.Mode, LADDR := #Diagnostic10.ET_200SP.RelaySafety_10.LADDR, DIAG := #Diagnostic10.ET_200SP.RelaySafety_10.diagDIS, DETAIL :=, RET_VAL => #Diagnostic10.ET_200SP.RelaySafety_10.RetVal, CNT_DIAG => #Diagnostic10.ET_200SP.RelaySafety_10.cntDiag)
   END_RUNG
   // the same network as SCL:
   #Diagnostic10.ET_200SP.RelaySafety_10.RetVal := GET_DIAG(MODE := #Diagnostic10.ET_200SP.RelaySafety_10.Mode,
                           LADDR := #Diagnostic10.ET_200SP.RelaySafety_10.LADDR,
                           DIAG := #Diagnostic10.ET_200SP.RelaySafety_10.diagDIS,
                           CNT_DIAG => #Diagnostic10.ET_200SP.RelaySafety_10.cntDiag);
END_REGION

REGION Network 24
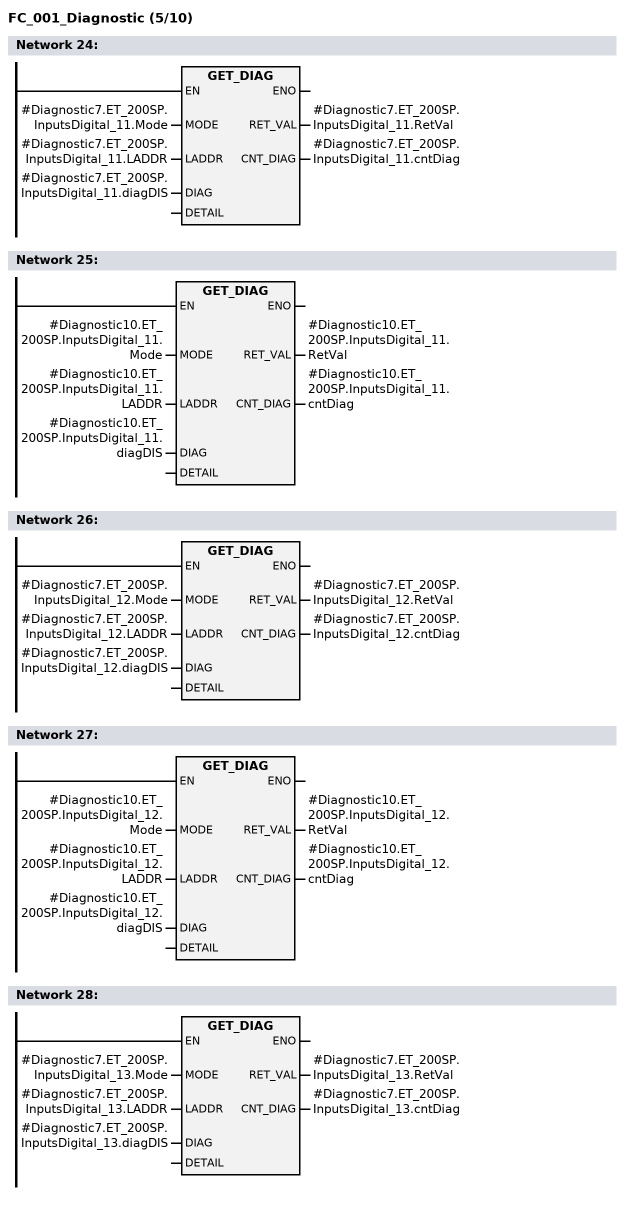
   RUNG wire#powerrail
      GET_DIAG(MODE := #Diagnostic7.ET_200SP.InputsDigital_11.Mode, LADDR := #Diagnostic7.ET_200SP.InputsDigital_11.LADDR, DIAG := #Diagnostic7.ET_200SP.InputsDigital_11.diagDIS, DETAIL :=, RET_VAL => #Diagnostic7.ET_200SP.InputsDigital_11.RetVal, CNT_DIAG => #Diagnostic7.ET_200SP.InputsDigital_11.cntDiag)
   END_RUNG
   // the same network as SCL:
   #Diagnostic7.ET_200SP.InputsDigital_11.RetVal := GET_DIAG(MODE := #Diagnostic7.ET_200SP.InputsDigital_11.Mode,
                           LADDR := #Diagnostic7.ET_200SP.InputsDigital_11.LADDR,
                           DIAG := #Diagnostic7.ET_200SP.InputsDigital_11.diagDIS,
                           CNT_DIAG => #Diagnostic7.ET_200SP.InputsDigital_11.cntDiag);
END_REGION

REGION Network 25
   RUNG wire#powerrail
      GET_DIAG(MODE := #Diagnostic10.ET_200SP.InputsDigital_11.Mode, LADDR := #Diagnostic10.ET_200SP.InputsDigital_11.LADDR, DIAG := #Diagnostic10.ET_200SP.InputsDigital_11.diagDIS, DETAIL :=, RET_VAL => #Diagnostic10.ET_200SP.InputsDigital_11.RetVal, CNT_DIAG => #Diagnostic10.ET_200SP.InputsDigital_11.cntDiag)
   END_RUNG
   // the same network as SCL:
   #Diagnostic10.ET_200SP.InputsDigital_11.RetVal := GET_DIAG(MODE := #Diagnostic10.ET_200SP.InputsDigital_11.Mode,
                           LADDR := #Diagnostic10.ET_200SP.InputsDigital_11.LADDR,
                           DIAG := #Diagnostic10.ET_200SP.InputsDigital_11.diagDIS,
                           CNT_DIAG => #Diagnostic10.ET_200SP.InputsDigital_11.cntDiag);
END_REGION

REGION Network 26
   RUNG wire#powerrail
      GET_DIAG(MODE := #Diagnostic7.ET_200SP.InputsDigital_12.Mode, LADDR := #Diagnostic7.ET_200SP.InputsDigital_12.LADDR, DIAG := #Diagnostic7.ET_200SP.InputsDigital_12.diagDIS, DETAIL :=, RET_VAL => #Diagnostic7.ET_200SP.InputsDigital_12.RetVal, CNT_DIAG => #Diagnostic7.ET_200SP.InputsDigital_12.cntDiag)
   END_RUNG
   // the same network as SCL:
   #Diagnostic7.ET_200SP.InputsDigital_12.RetVal := GET_DIAG(MODE := #Diagnostic7.ET_200SP.InputsDigital_12.Mode,
                           LADDR := #Diagnostic7.ET_200SP.InputsDigital_12.LADDR,
                           DIAG := #Diagnostic7.ET_200SP.InputsDigital_12.diagDIS,
                           CNT_DIAG => #Diagnostic7.ET_200SP.InputsDigital_12.cntDiag);
END_REGION

REGION Network 27
   RUNG wire#powerrail
      GET_DIAG(MODE := #Diagnostic10.ET_200SP.InputsDigital_12.Mode, LADDR := #Diagnostic10.ET_200SP.InputsDigital_12.LADDR, DIAG := #Diagnostic10.ET_200SP.InputsDigital_12.diagDIS, DETAIL :=, RET_VAL => #Diagnostic10.ET_200SP.InputsDigital_12.RetVal, CNT_DIAG => #Diagnostic10.ET_200SP.InputsDigital_12.cntDiag)
   END_RUNG
   // the same network as SCL:
   #Diagnostic10.ET_200SP.InputsDigital_12.RetVal := GET_DIAG(MODE := #Diagnostic10.ET_200SP.InputsDigital_12.Mode,
                           LADDR := #Diagnostic10.ET_200SP.InputsDigital_12.LADDR,
                           DIAG := #Diagnostic10.ET_200SP.InputsDigital_12.diagDIS,
                           CNT_DIAG => #Diagnostic10.ET_200SP.InputsDigital_12.cntDiag);
END_REGION

REGION Network 28
   RUNG wire#powerrail
      GET_DIAG(MODE := #Diagnostic7.ET_200SP.InputsDigital_13.Mode, LADDR := #Diagnostic7.ET_200SP.InputsDigital_13.LADDR, DIAG := #Diagnostic7.ET_200SP.InputsDigital_13.diagDIS, DETAIL :=, RET_VAL => #Diagnostic7.ET_200SP.InputsDigital_13.RetVal, CNT_DIAG => #Diagnostic7.ET_200SP.InputsDigital_13.cntDiag)
   END_RUNG
   // the same network as SCL:
   #Diagnostic7.ET_200SP.InputsDigital_13.RetVal := GET_DIAG(MODE := #Diagnostic7.ET_200SP.InputsDigital_13.Mode,
                           LADDR := #Diagnostic7.ET_200SP.InputsDigital_13.LADDR,
                           DIAG := #Diagnostic7.ET_200SP.InputsDigital_13.diagDIS,
                           CNT_DIAG => #Diagnostic7.ET_200SP.InputsDigital_13.cntDiag);
END_REGION

REGION Network 29
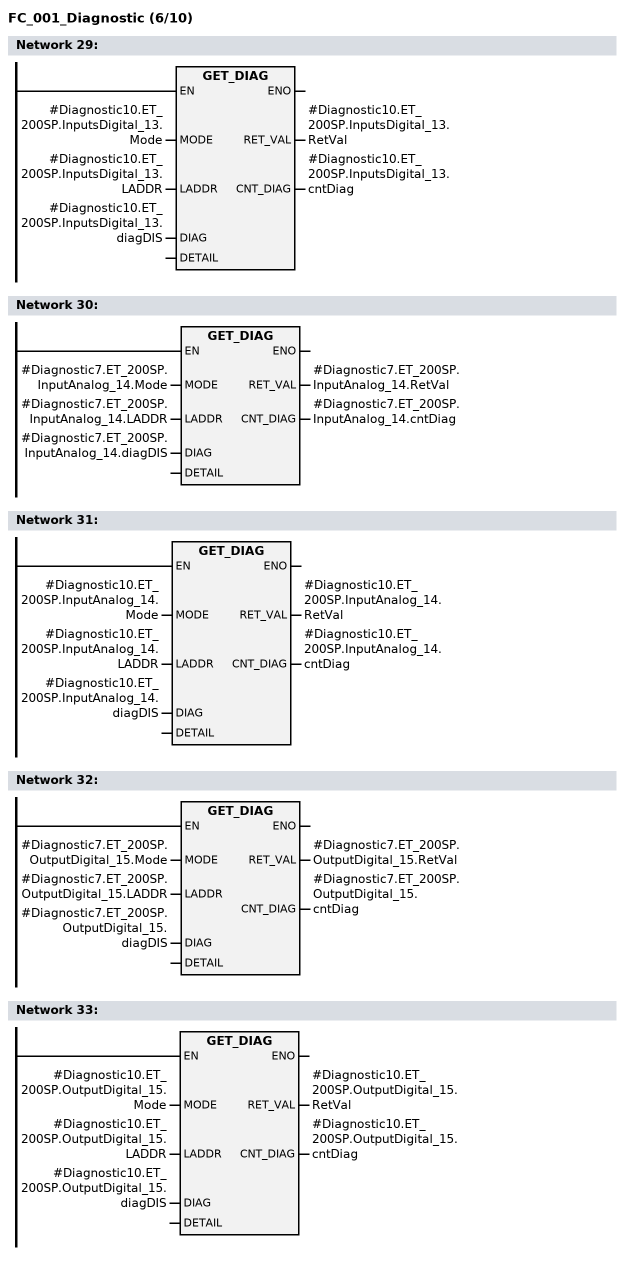
   RUNG wire#powerrail
      GET_DIAG(MODE := #Diagnostic10.ET_200SP.InputsDigital_13.Mode, LADDR := #Diagnostic10.ET_200SP.InputsDigital_13.LADDR, DIAG := #Diagnostic10.ET_200SP.InputsDigital_13.diagDIS, DETAIL :=, RET_VAL => #Diagnostic10.ET_200SP.InputsDigital_13.RetVal, CNT_DIAG => #Diagnostic10.ET_200SP.InputsDigital_13.cntDiag)
   END_RUNG
   // the same network as SCL:
   #Diagnostic10.ET_200SP.InputsDigital_13.RetVal := GET_DIAG(MODE := #Diagnostic10.ET_200SP.InputsDigital_13.Mode,
                           LADDR := #Diagnostic10.ET_200SP.InputsDigital_13.LADDR,
                           DIAG := #Diagnostic10.ET_200SP.InputsDigital_13.diagDIS,
                           CNT_DIAG => #Diagnostic10.ET_200SP.InputsDigital_13.cntDiag);
END_REGION

REGION Network 30
   RUNG wire#powerrail
      GET_DIAG(MODE := #Diagnostic7.ET_200SP.InputAnalog_14.Mode, LADDR := #Diagnostic7.ET_200SP.InputAnalog_14.LADDR, DIAG := #Diagnostic7.ET_200SP.InputAnalog_14.diagDIS, DETAIL :=, RET_VAL => #Diagnostic7.ET_200SP.InputAnalog_14.RetVal, CNT_DIAG => #Diagnostic7.ET_200SP.InputAnalog_14.cntDiag)
   END_RUNG
   // the same network as SCL:
   #Diagnostic7.ET_200SP.InputAnalog_14.RetVal := GET_DIAG(MODE := #Diagnostic7.ET_200SP.InputAnalog_14.Mode,
                           LADDR := #Diagnostic7.ET_200SP.InputAnalog_14.LADDR,
                           DIAG := #Diagnostic7.ET_200SP.InputAnalog_14.diagDIS,
                           CNT_DIAG => #Diagnostic7.ET_200SP.InputAnalog_14.cntDiag);
END_REGION

REGION Network 31
   RUNG wire#powerrail
      GET_DIAG(MODE := #Diagnostic10.ET_200SP.InputAnalog_14.Mode, LADDR := #Diagnostic10.ET_200SP.InputAnalog_14.LADDR, DIAG := #Diagnostic10.ET_200SP.InputAnalog_14.diagDIS, DETAIL :=, RET_VAL => #Diagnostic10.ET_200SP.InputAnalog_14.RetVal, CNT_DIAG => #Diagnostic10.ET_200SP.InputAnalog_14.cntDiag)
   END_RUNG
   // the same network as SCL:
   #Diagnostic10.ET_200SP.InputAnalog_14.RetVal := GET_DIAG(MODE := #Diagnostic10.ET_200SP.InputAnalog_14.Mode,
                           LADDR := #Diagnostic10.ET_200SP.InputAnalog_14.LADDR,
                           DIAG := #Diagnostic10.ET_200SP.InputAnalog_14.diagDIS,
                           CNT_DIAG => #Diagnostic10.ET_200SP.InputAnalog_14.cntDiag);
END_REGION

REGION Network 32
   RUNG wire#powerrail
      GET_DIAG(MODE := #Diagnostic7.ET_200SP.OutputDigital_15.Mode, LADDR := #Diagnostic7.ET_200SP.OutputDigital_15.LADDR, DIAG := #Diagnostic7.ET_200SP.OutputDigital_15.diagDIS, DETAIL :=, RET_VAL => #Diagnostic7.ET_200SP.OutputDigital_15.RetVal, CNT_DIAG => #Diagnostic7.ET_200SP.OutputDigital_15.cntDiag)
   END_RUNG
   // the same network as SCL:
   #Diagnostic7.ET_200SP.OutputDigital_15.RetVal := GET_DIAG(MODE := #Diagnostic7.ET_200SP.OutputDigital_15.Mode,
                           LADDR := #Diagnostic7.ET_200SP.OutputDigital_15.LADDR,
                           DIAG := #Diagnostic7.ET_200SP.OutputDigital_15.diagDIS,
                           CNT_DIAG => #Diagnostic7.ET_200SP.OutputDigital_15.cntDiag);
END_REGION

REGION Network 33
   RUNG wire#powerrail
      GET_DIAG(MODE := #Diagnostic10.ET_200SP.OutputDigital_15.Mode, LADDR := #Diagnostic10.ET_200SP.OutputDigital_15.LADDR, DIAG := #Diagnostic10.ET_200SP.OutputDigital_15.diagDIS, DETAIL :=, RET_VAL => #Diagnostic10.ET_200SP.OutputDigital_15.RetVal, CNT_DIAG => #Diagnostic10.ET_200SP.OutputDigital_15.cntDiag)
   END_RUNG
   // the same network as SCL:
   #Diagnostic10.ET_200SP.OutputDigital_15.RetVal := GET_DIAG(MODE := #Diagnostic10.ET_200SP.OutputDigital_15.Mode,
                           LADDR := #Diagnostic10.ET_200SP.OutputDigital_15.LADDR,
                           DIAG := #Diagnostic10.ET_200SP.OutputDigital_15.diagDIS,
                           CNT_DIAG => #Diagnostic10.ET_200SP.OutputDigital_15.cntDiag);
END_REGION

REGION Network 34
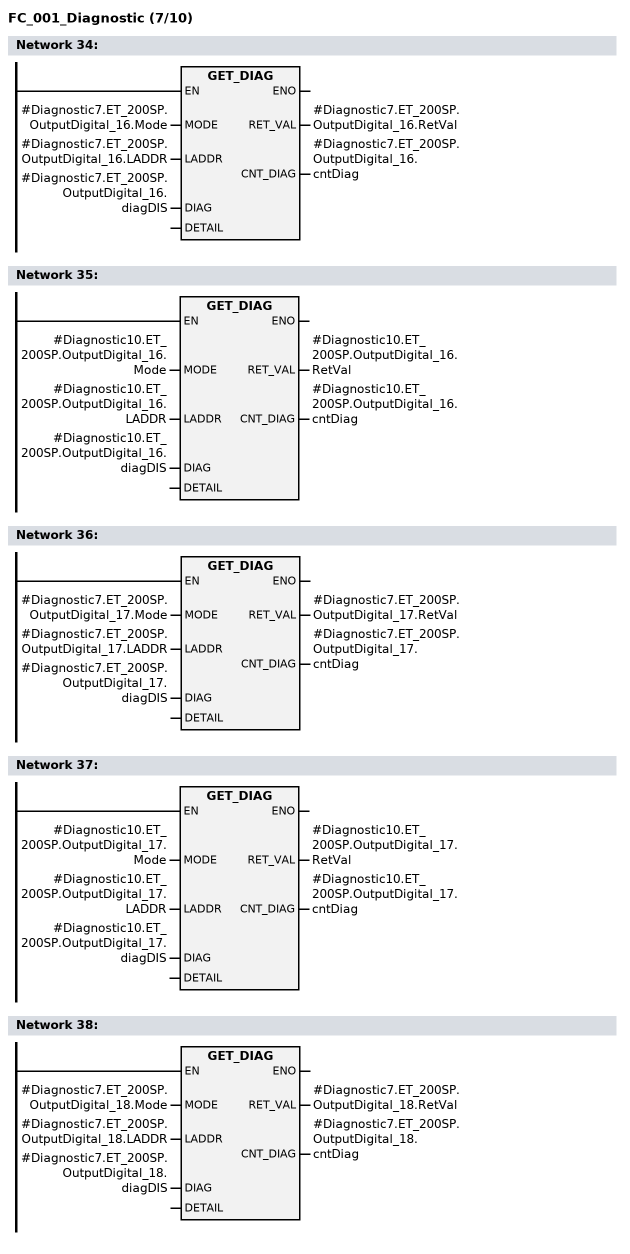
   RUNG wire#powerrail
      GET_DIAG(MODE := #Diagnostic7.ET_200SP.OutputDigital_16.Mode, LADDR := #Diagnostic7.ET_200SP.OutputDigital_16.LADDR, DIAG := #Diagnostic7.ET_200SP.OutputDigital_16.diagDIS, DETAIL :=, RET_VAL => #Diagnostic7.ET_200SP.OutputDigital_16.RetVal, CNT_DIAG => #Diagnostic7.ET_200SP.OutputDigital_16.cntDiag)
   END_RUNG
   // the same network as SCL:
   #Diagnostic7.ET_200SP.OutputDigital_16.RetVal := GET_DIAG(MODE := #Diagnostic7.ET_200SP.OutputDigital_16.Mode,
                           LADDR := #Diagnostic7.ET_200SP.OutputDigital_16.LADDR,
                           DIAG := #Diagnostic7.ET_200SP.OutputDigital_16.diagDIS,
                           CNT_DIAG => #Diagnostic7.ET_200SP.OutputDigital_16.cntDiag);
END_REGION

REGION Network 35
   RUNG wire#powerrail
      GET_DIAG(MODE := #Diagnostic10.ET_200SP.OutputDigital_16.Mode, LADDR := #Diagnostic10.ET_200SP.OutputDigital_16.LADDR, DIAG := #Diagnostic10.ET_200SP.OutputDigital_16.diagDIS, DETAIL :=, RET_VAL => #Diagnostic10.ET_200SP.OutputDigital_16.RetVal, CNT_DIAG => #Diagnostic10.ET_200SP.OutputDigital_16.cntDiag)
   END_RUNG
   // the same network as SCL:
   #Diagnostic10.ET_200SP.OutputDigital_16.RetVal := GET_DIAG(MODE := #Diagnostic10.ET_200SP.OutputDigital_16.Mode,
                           LADDR := #Diagnostic10.ET_200SP.OutputDigital_16.LADDR,
                           DIAG := #Diagnostic10.ET_200SP.OutputDigital_16.diagDIS,
                           CNT_DIAG => #Diagnostic10.ET_200SP.OutputDigital_16.cntDiag);
END_REGION

REGION Network 36
   RUNG wire#powerrail
      GET_DIAG(MODE := #Diagnostic7.ET_200SP.OutputDigital_17.Mode, LADDR := #Diagnostic7.ET_200SP.OutputDigital_17.LADDR, DIAG := #Diagnostic7.ET_200SP.OutputDigital_17.diagDIS, DETAIL :=, RET_VAL => #Diagnostic7.ET_200SP.OutputDigital_17.RetVal, CNT_DIAG => #Diagnostic7.ET_200SP.OutputDigital_17.cntDiag)
   END_RUNG
   // the same network as SCL:
   #Diagnostic7.ET_200SP.OutputDigital_17.RetVal := GET_DIAG(MODE := #Diagnostic7.ET_200SP.OutputDigital_17.Mode,
                           LADDR := #Diagnostic7.ET_200SP.OutputDigital_17.LADDR,
                           DIAG := #Diagnostic7.ET_200SP.OutputDigital_17.diagDIS,
                           CNT_DIAG => #Diagnostic7.ET_200SP.OutputDigital_17.cntDiag);
END_REGION

REGION Network 37
   RUNG wire#powerrail
      GET_DIAG(MODE := #Diagnostic10.ET_200SP.OutputDigital_17.Mode, LADDR := #Diagnostic10.ET_200SP.OutputDigital_17.LADDR, DIAG := #Diagnostic10.ET_200SP.OutputDigital_17.diagDIS, DETAIL :=, RET_VAL => #Diagnostic10.ET_200SP.OutputDigital_17.RetVal, CNT_DIAG => #Diagnostic10.ET_200SP.OutputDigital_17.cntDiag)
   END_RUNG
   // the same network as SCL:
   #Diagnostic10.ET_200SP.OutputDigital_17.RetVal := GET_DIAG(MODE := #Diagnostic10.ET_200SP.OutputDigital_17.Mode,
                           LADDR := #Diagnostic10.ET_200SP.OutputDigital_17.LADDR,
                           DIAG := #Diagnostic10.ET_200SP.OutputDigital_17.diagDIS,
                           CNT_DIAG => #Diagnostic10.ET_200SP.OutputDigital_17.cntDiag);
END_REGION

REGION Network 38
   RUNG wire#powerrail
      GET_DIAG(MODE := #Diagnostic7.ET_200SP.OutputDigital_18.Mode, LADDR := #Diagnostic7.ET_200SP.OutputDigital_18.LADDR, DIAG := #Diagnostic7.ET_200SP.OutputDigital_18.diagDIS, DETAIL :=, RET_VAL => #Diagnostic7.ET_200SP.OutputDigital_18.RetVal, CNT_DIAG => #Diagnostic7.ET_200SP.OutputDigital_18.cntDiag)
   END_RUNG
   // the same network as SCL:
   #Diagnostic7.ET_200SP.OutputDigital_18.RetVal := GET_DIAG(MODE := #Diagnostic7.ET_200SP.OutputDigital_18.Mode,
                           LADDR := #Diagnostic7.ET_200SP.OutputDigital_18.LADDR,
                           DIAG := #Diagnostic7.ET_200SP.OutputDigital_18.diagDIS,
                           CNT_DIAG => #Diagnostic7.ET_200SP.OutputDigital_18.cntDiag);
END_REGION

REGION Network 39
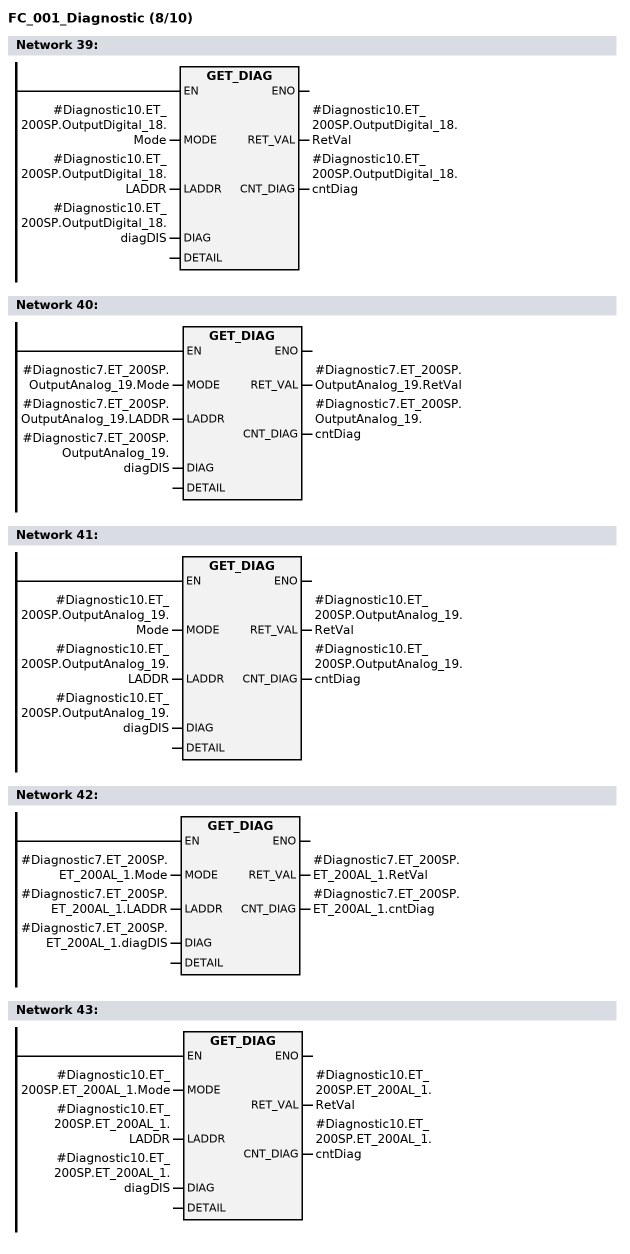
   RUNG wire#powerrail
      GET_DIAG(MODE := #Diagnostic10.ET_200SP.OutputDigital_18.Mode, LADDR := #Diagnostic10.ET_200SP.OutputDigital_18.LADDR, DIAG := #Diagnostic10.ET_200SP.OutputDigital_18.diagDIS, DETAIL :=, RET_VAL => #Diagnostic10.ET_200SP.OutputDigital_18.RetVal, CNT_DIAG => #Diagnostic10.ET_200SP.OutputDigital_18.cntDiag)
   END_RUNG
   // the same network as SCL:
   #Diagnostic10.ET_200SP.OutputDigital_18.RetVal := GET_DIAG(MODE := #Diagnostic10.ET_200SP.OutputDigital_18.Mode,
                           LADDR := #Diagnostic10.ET_200SP.OutputDigital_18.LADDR,
                           DIAG := #Diagnostic10.ET_200SP.OutputDigital_18.diagDIS,
                           CNT_DIAG => #Diagnostic10.ET_200SP.OutputDigital_18.cntDiag);
END_REGION

REGION Network 40
   RUNG wire#powerrail
      GET_DIAG(MODE := #Diagnostic7.ET_200SP.OutputAnalog_19.Mode, LADDR := #Diagnostic7.ET_200SP.OutputAnalog_19.LADDR, DIAG := #Diagnostic7.ET_200SP.OutputAnalog_19.diagDIS, DETAIL :=, RET_VAL => #Diagnostic7.ET_200SP.OutputAnalog_19.RetVal, CNT_DIAG => #Diagnostic7.ET_200SP.OutputAnalog_19.cntDiag)
   END_RUNG
   // the same network as SCL:
   #Diagnostic7.ET_200SP.OutputAnalog_19.RetVal := GET_DIAG(MODE := #Diagnostic7.ET_200SP.OutputAnalog_19.Mode,
                           LADDR := #Diagnostic7.ET_200SP.OutputAnalog_19.LADDR,
                           DIAG := #Diagnostic7.ET_200SP.OutputAnalog_19.diagDIS,
                           CNT_DIAG => #Diagnostic7.ET_200SP.OutputAnalog_19.cntDiag);
END_REGION

REGION Network 41
   RUNG wire#powerrail
      GET_DIAG(MODE := #Diagnostic10.ET_200SP.OutputAnalog_19.Mode, LADDR := #Diagnostic10.ET_200SP.OutputAnalog_19.LADDR, DIAG := #Diagnostic10.ET_200SP.OutputAnalog_19.diagDIS, DETAIL :=, RET_VAL => #Diagnostic10.ET_200SP.OutputAnalog_19.RetVal, CNT_DIAG => #Diagnostic10.ET_200SP.OutputAnalog_19.cntDiag)
   END_RUNG
   // the same network as SCL:
   #Diagnostic10.ET_200SP.OutputAnalog_19.RetVal := GET_DIAG(MODE := #Diagnostic10.ET_200SP.OutputAnalog_19.Mode,
                           LADDR := #Diagnostic10.ET_200SP.OutputAnalog_19.LADDR,
                           DIAG := #Diagnostic10.ET_200SP.OutputAnalog_19.diagDIS,
                           CNT_DIAG => #Diagnostic10.ET_200SP.OutputAnalog_19.cntDiag);
END_REGION

REGION Network 42
   RUNG wire#powerrail
      GET_DIAG(MODE := #Diagnostic7.ET_200SP.ET_200AL_1.Mode, LADDR := #Diagnostic7.ET_200SP.ET_200AL_1.LADDR, DIAG := #Diagnostic7.ET_200SP.ET_200AL_1.diagDIS, DETAIL :=, RET_VAL => #Diagnostic7.ET_200SP.ET_200AL_1.RetVal, CNT_DIAG => #Diagnostic7.ET_200SP.ET_200AL_1.cntDiag)
   END_RUNG
   // the same network as SCL:
   #Diagnostic7.ET_200SP.ET_200AL_1.RetVal := GET_DIAG(MODE := #Diagnostic7.ET_200SP.ET_200AL_1.Mode,
                           LADDR := #Diagnostic7.ET_200SP.ET_200AL_1.LADDR,
                           DIAG := #Diagnostic7.ET_200SP.ET_200AL_1.diagDIS,
                           CNT_DIAG => #Diagnostic7.ET_200SP.ET_200AL_1.cntDiag);
END_REGION

REGION Network 43
   RUNG wire#powerrail
      GET_DIAG(MODE := #Diagnostic10.ET_200SP.ET_200AL_1.Mode, LADDR := #Diagnostic10.ET_200SP.ET_200AL_1.LADDR, DIAG := #Diagnostic10.ET_200SP.ET_200AL_1.diagDIS, DETAIL :=, RET_VAL => #Diagnostic10.ET_200SP.ET_200AL_1.RetVal, CNT_DIAG => #Diagnostic10.ET_200SP.ET_200AL_1.cntDiag)
   END_RUNG
   // the same network as SCL:
   #Diagnostic10.ET_200SP.ET_200AL_1.RetVal := GET_DIAG(MODE := #Diagnostic10.ET_200SP.ET_200AL_1.Mode,
                           LADDR := #Diagnostic10.ET_200SP.ET_200AL_1.LADDR,
                           DIAG := #Diagnostic10.ET_200SP.ET_200AL_1.diagDIS,
                           CNT_DIAG => #Diagnostic10.ET_200SP.ET_200AL_1.cntDiag);
END_REGION

REGION Network 44
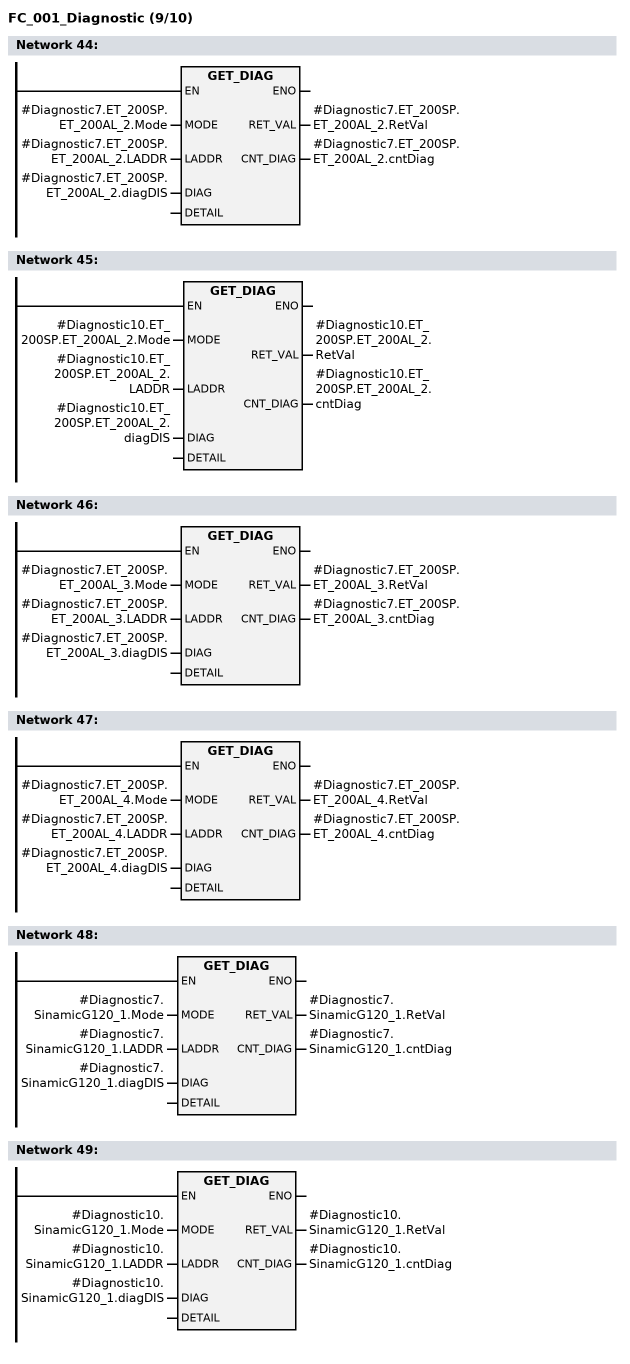
   RUNG wire#powerrail
      GET_DIAG(MODE := #Diagnostic7.ET_200SP.ET_200AL_2.Mode, LADDR := #Diagnostic7.ET_200SP.ET_200AL_2.LADDR, DIAG := #Diagnostic7.ET_200SP.ET_200AL_2.diagDIS, DETAIL :=, RET_VAL => #Diagnostic7.ET_200SP.ET_200AL_2.RetVal, CNT_DIAG => #Diagnostic7.ET_200SP.ET_200AL_2.cntDiag)
   END_RUNG
   // the same network as SCL:
   #Diagnostic7.ET_200SP.ET_200AL_2.RetVal := GET_DIAG(MODE := #Diagnostic7.ET_200SP.ET_200AL_2.Mode,
                           LADDR := #Diagnostic7.ET_200SP.ET_200AL_2.LADDR,
                           DIAG := #Diagnostic7.ET_200SP.ET_200AL_2.diagDIS,
                           CNT_DIAG => #Diagnostic7.ET_200SP.ET_200AL_2.cntDiag);
END_REGION

REGION Network 45
   RUNG wire#powerrail
      GET_DIAG(MODE := #Diagnostic10.ET_200SP.ET_200AL_2.Mode, LADDR := #Diagnostic10.ET_200SP.ET_200AL_2.LADDR, DIAG := #Diagnostic10.ET_200SP.ET_200AL_2.diagDIS, DETAIL :=, RET_VAL => #Diagnostic10.ET_200SP.ET_200AL_2.RetVal, CNT_DIAG => #Diagnostic10.ET_200SP.ET_200AL_2.cntDiag)
   END_RUNG
   // the same network as SCL:
   #Diagnostic10.ET_200SP.ET_200AL_2.RetVal := GET_DIAG(MODE := #Diagnostic10.ET_200SP.ET_200AL_2.Mode,
                           LADDR := #Diagnostic10.ET_200SP.ET_200AL_2.LADDR,
                           DIAG := #Diagnostic10.ET_200SP.ET_200AL_2.diagDIS,
                           CNT_DIAG => #Diagnostic10.ET_200SP.ET_200AL_2.cntDiag);
END_REGION

REGION Network 46
   RUNG wire#powerrail
      GET_DIAG(MODE := #Diagnostic7.ET_200SP.ET_200AL_3.Mode, LADDR := #Diagnostic7.ET_200SP.ET_200AL_3.LADDR, DIAG := #Diagnostic7.ET_200SP.ET_200AL_3.diagDIS, DETAIL :=, RET_VAL => #Diagnostic7.ET_200SP.ET_200AL_3.RetVal, CNT_DIAG => #Diagnostic7.ET_200SP.ET_200AL_3.cntDiag)
   END_RUNG
   // the same network as SCL:
   #Diagnostic7.ET_200SP.ET_200AL_3.RetVal := GET_DIAG(MODE := #Diagnostic7.ET_200SP.ET_200AL_3.Mode,
                           LADDR := #Diagnostic7.ET_200SP.ET_200AL_3.LADDR,
                           DIAG := #Diagnostic7.ET_200SP.ET_200AL_3.diagDIS,
                           CNT_DIAG => #Diagnostic7.ET_200SP.ET_200AL_3.cntDiag);
END_REGION

REGION Network 47
   RUNG wire#powerrail
      GET_DIAG(MODE := #Diagnostic7.ET_200SP.ET_200AL_4.Mode, LADDR := #Diagnostic7.ET_200SP.ET_200AL_4.LADDR, DIAG := #Diagnostic7.ET_200SP.ET_200AL_4.diagDIS, DETAIL :=, RET_VAL => #Diagnostic7.ET_200SP.ET_200AL_4.RetVal, CNT_DIAG => #Diagnostic7.ET_200SP.ET_200AL_4.cntDiag)
   END_RUNG
   // the same network as SCL:
   #Diagnostic7.ET_200SP.ET_200AL_4.RetVal := GET_DIAG(MODE := #Diagnostic7.ET_200SP.ET_200AL_4.Mode,
                           LADDR := #Diagnostic7.ET_200SP.ET_200AL_4.LADDR,
                           DIAG := #Diagnostic7.ET_200SP.ET_200AL_4.diagDIS,
                           CNT_DIAG => #Diagnostic7.ET_200SP.ET_200AL_4.cntDiag);
END_REGION

REGION Network 48
   RUNG wire#powerrail
      GET_DIAG(MODE := #Diagnostic7.SinamicG120_1.Mode, LADDR := #Diagnostic7.SinamicG120_1.LADDR, DIAG := #Diagnostic7.SinamicG120_1.diagDIS, DETAIL :=, RET_VAL => #Diagnostic7.SinamicG120_1.RetVal, CNT_DIAG => #Diagnostic7.SinamicG120_1.cntDiag)
   END_RUNG
   // the same network as SCL:
   #Diagnostic7.SinamicG120_1.RetVal := GET_DIAG(MODE := #Diagnostic7.SinamicG120_1.Mode,
                           LADDR := #Diagnostic7.SinamicG120_1.LADDR,
                           DIAG := #Diagnostic7.SinamicG120_1.diagDIS,
                           CNT_DIAG => #Diagnostic7.SinamicG120_1.cntDiag);
END_REGION

REGION Network 49
   RUNG wire#powerrail
      GET_DIAG(MODE := #Diagnostic10.SinamicG120_1.Mode, LADDR := #Diagnostic10.SinamicG120_1.LADDR, DIAG := #Diagnostic10.SinamicG120_1.diagDIS, DETAIL :=, RET_VAL => #Diagnostic10.SinamicG120_1.RetVal, CNT_DIAG => #Diagnostic10.SinamicG120_1.cntDiag)
   END_RUNG
   // the same network as SCL:
   #Diagnostic10.SinamicG120_1.RetVal := GET_DIAG(MODE := #Diagnostic10.SinamicG120_1.Mode,
                           LADDR := #Diagnostic10.SinamicG120_1.LADDR,
                           DIAG := #Diagnostic10.SinamicG120_1.diagDIS,
                           CNT_DIAG => #Diagnostic10.SinamicG120_1.cntDiag);
END_REGION

REGION Network 50
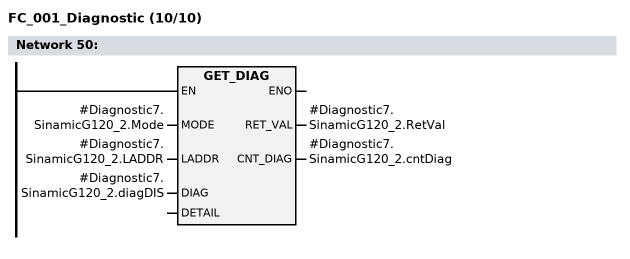
   RUNG wire#powerrail
      GET_DIAG(MODE := #Diagnostic7.SinamicG120_2.Mode, LADDR := #Diagnostic7.SinamicG120_2.LADDR, DIAG := #Diagnostic7.SinamicG120_2.diagDIS, DETAIL :=, RET_VAL => #Diagnostic7.SinamicG120_2.RetVal, CNT_DIAG => #Diagnostic7.SinamicG120_2.cntDiag)
   END_RUNG
   // the same network as SCL:
   #Diagnostic7.SinamicG120_2.RetVal := GET_DIAG(MODE := #Diagnostic7.SinamicG120_2.Mode,
                           LADDR := #Diagnostic7.SinamicG120_2.LADDR,
                           DIAG := #Diagnostic7.SinamicG120_2.diagDIS,
                           CNT_DIAG => #Diagnostic7.SinamicG120_2.cntDiag);
END_REGION

REGION Network 51 (SCL)
   // Diagnostyka dla szafy 1
   #Diagnostic7.DiagnosticOK := #Diagnostic7.ET_200SP.HeadModule_0.diagDIS.OwnState = 0 AND
   #Diagnostic7.ET_200SP.BusAdapter_1.diagDIS.OwnState = 0 AND #Diagnostic7.ET_200SP.InputSafety_2.diagDIS.OwnState = 0 AND
   #Diagnostic7.ET_200SP.InputSafety_3.diagDIS.OwnState = 0 AND #Diagnostic7.ET_200SP.InputSafety_4.diagDIS.OwnState = 0 AND
   #Diagnostic7.ET_200SP.InputSafety_5.diagDIS.OwnState = 0 AND #Diagnostic7.ET_200SP.OutputSafety_7.diagDIS.OwnState = 0 AND
   #Diagnostic7.ET_200SP.RelaySafety_9.diagDIS.OwnState = 0 AND #Diagnostic7.ET_200SP.InputSafety_6.diagDIS.OwnState = 0 AND
   #Diagnostic7.ET_200SP.RelaySafety_10.diagDIS.OwnState = 0 AND #Diagnostic7.ET_200SP.InputsDigital_11.diagDIS.OwnState = 0 AND
   #Diagnostic7.ET_200SP.InputsDigital_12.diagDIS.OwnState = 0 AND #Diagnostic7.ET_200SP.InputsDigital_13.diagDIS.OwnState = 0 AND
   #Diagnostic7.ET_200SP.InputAnalog_14.diagDIS.OwnState = 0 AND #Diagnostic7.ET_200SP.OutputDigital_15.diagDIS.OwnState = 0 AND
   #Diagnostic7.ET_200SP.OutputDigital_16.diagDIS.OwnState = 0 AND #Diagnostic7.ET_200SP.OutputDigital_17.diagDIS.OwnState = 0 AND
   #Diagnostic7.ET_200SP.OutputDigital_18.diagDIS.OwnState = 0 AND #Diagnostic7.ET_200SP.OutputAnalog_19.diagDIS.OwnState = 0 AND
   #Diagnostic7.ET_200SP.ET_200AL_1.diagDIS.OwnState = 0 AND #Diagnostic7.ET_200SP.ET_200AL_2.diagDIS.OwnState = 0 AND
   #Diagnostic7.ET_200SP.ET_200AL_3.diagDIS.OwnState = 0 AND #Diagnostic7.ET_200SP.ET_200AL_4.diagDIS.OwnState = 0 AND
   #Diagnostic7.SinamicG120_1.diagDIS.OwnState = 0 AND #Diagnostic7.SinamicG120_2.diagDIS.OwnState = 0;
END_REGION

REGION Network 52 (SCL)
   //DIAGNOSTYKA 10 
   #Diagnostic10.DiagnosticOK := #Diagnostic10.ET_200SP.HeadModule_0.diagDIS.OwnState = 0 AND
   #Diagnostic10.ET_200SP.BusAdapter_1.diagDIS.OwnState = 0 AND #Diagnostic10.ET_200SP.InputSafety_2.diagDIS.OwnState = 0 AND
   #Diagnostic10.ET_200SP.InputSafety_3.diagDIS.OwnState = 0 AND #Diagnostic10.ET_200SP.InputSafety_4.diagDIS.OwnState = 0 AND
   #Diagnostic10.ET_200SP.InputSafety_5.diagDIS.OwnState = 0 AND #Diagnostic10.ET_200SP.OutputSafety_7.diagDIS.OwnState = 0 AND
   #Diagnostic10.ET_200SP.RelaySafety_9.diagDIS.OwnState = 0 AND #Diagnostic10.ET_200SP.InputSafety_6.diagDIS.OwnState = 0 AND
   #Diagnostic10.ET_200SP.RelaySafety_10.diagDIS.OwnState = 0 AND #Diagnostic10.ET_200SP.InputsDigital_11.diagDIS.OwnState = 0 AND
   #Diagnostic10.ET_200SP.InputsDigital_12.diagDIS.OwnState = 0 AND #Diagnostic10.ET_200SP.InputsDigital_13.diagDIS.OwnState = 0 AND
   #Diagnostic10.ET_200SP.InputAnalog_14.diagDIS.OwnState = 0 AND #Diagnostic10.ET_200SP.OutputDigital_15.diagDIS.OwnState = 0 AND
   #Diagnostic10.ET_200SP.OutputDigital_16.diagDIS.OwnState = 0 AND #Diagnostic10.ET_200SP.OutputDigital_17.diagDIS.OwnState = 0 AND
   #Diagnostic10.ET_200SP.OutputDigital_18.diagDIS.OwnState = 0 AND #Diagnostic10.ET_200SP.OutputAnalog_19.diagDIS.OwnState = 0 AND
   #Diagnostic10.ET_200SP.ET_200AL_1.diagDIS.OwnState = 0 AND #Diagnostic10.ET_200SP.ET_200AL_2.diagDIS.OwnState = 0 AND
   #Diagnostic10.SinamicG120_1.diagDIS.OwnState = 0;
END_REGION
END_FUNCTION

FUNCTION "FC_002_Inputs&Recipe" : Void
{ S7_Optimized_Access := 'TRUE' }
VERSION : 0.1

BEGIN
	//************************************************************
	//===Author: Mateusz Połojko
	//-----Linkedin: https://pl.linkedin.com/in/mateusz-po%C5%82ojko-52a3541b1
	//-----Github: https://github.com/Bhazel95
	//===Description:
	//-----Hardware input assigment & Recipes
	//===Customer:
	//-----Apator Powogaz S.A.
	//************************************************************
	
	REGION 7A
	    REGION Button box left
	        "DEV_7".Convoyer.Modular_A.ButtonControl.ButtonBoxLeft.ButtonReset := "7A_BUTTON_RESET_1";
	        "DEV_7".Convoyer.Modular_A.ButtonControl.ButtonBoxLeft.ButtonStart := "7A_BUTTON_START_1";
	        "DEV_7".Convoyer.Modular_A.ButtonControl.ButtonBoxLeft.ButtonStop := "7A_BUTTON_STOP_1";
	        "DEV_7".Convoyer.Modular_A.Safety.ESTOP_Left := "7A_ESTOP_1";
	    END_REGION
	    REGION Button box right
	        "DEV_7".Convoyer.Modular_A.ButtonControl.ButtonBoxRight.ButtonReset := "7A_BUTTON_RESET_2";
	        "DEV_7".Convoyer.Modular_A.ButtonControl.ButtonBoxRight.ButtonStart := "7A_BUTTON_START_2";
	        "DEV_7".Convoyer.Modular_A.ButtonControl.ButtonBoxRight.ButtonStop := "7A_BUTTON_STOP_2";
	        "DEV_7".Convoyer.Modular_A.Safety.ESTOP_Right := "7A_ESTOP_2";
	    END_REGION
	    REGION Main Cabinet    
	        "DEV_7".Convoyer.Modular_A.ButtonControl.CabinetBox.ButtonReset := "7_BUTTON_RESET";
	        "DEV_7".Convoyer.Modular_A.Safety.ESTOP_MAIN := "7_ESTOP";
	    END_REGION
	    REGION Pneumatics
	        "DEV_7".Convoyer.Modular_A.Pneumatics.Stamping.Sensors.In := "7A_ActuatorIn";
	        "DEV_7".Convoyer.Modular_A.Pneumatics.Stamping.Sensors.Out := "7A_ActuatorOut";
	        "DEV_7".Convoyer.Modular_A.Pneumatics.IVT.Sensor.Analog.RealValue := "7A_IVT_InputSignal_1";
	        "DEV_7".Convoyer.Modular_A.Pneumatics.IVT.Sensor.Scaled.RealNorm := NORM_X(MIN := 0, VALUE := "DEV_7".Convoyer.Modular_A.Pneumatics.IVT.Sensor.Analog.RealValue, MAX := 32767);
	        "DEV_7".Convoyer.Modular_A.Pneumatics.IVT.Sensor.Scaled.RealScale := SCALE_X(MIN := 0, VALUE := "DEV_7".Convoyer.Modular_A.Pneumatics.IVT.Sensor.Scaled.RealNorm, MAX := 7);
	    END_REGION
	    
	    REGION Sensors
	        "DEV_7".Convoyer.Modular_A.Sensors.Homing_I := "7A_Homing_I";
	        "DEV_7".Convoyer.Modular_A.Sensors.Homing_R := "7A_Homing_R";
	        "DEV_7".Convoyer.Modular_A.Sensors.StampingPresence := "7A_StampingPresence" AND "DEV_7".Convoyer.Modular_A.HMI.Stamping.Enable;
	        "DEV_7".Convoyer.Modular_A.Sensors.Stamp_Check_1 := "7A_StampingCheck_1";
	        "DEV_7".Convoyer.Modular_A.Sensors.Stamp_Check_2 := "7A_StampingCheck_2";
	        "DEV_7".Convoyer.Modular_A.Sensors.BlowPresence := "7A_BlowPresence";
	        "DEV_7".Convoyer.Modular_A.Sensors.CameraPresence := "7A_CameraPresence";
	        "DEV_7".Convoyer.Modular_A.Sensors.UnloadingPresence := "7A_UnloadingPresence";
	        "DEV_7".Convoyer.Modular_A.Sensors.Span := "7A_Span";
	        "DEV_7".Convoyer.Modular_A.Sensors.JogBack := "7A_JogBack";
	    END_REGION
	    
	    REGION Light curtains
	        "DEV_7".Convoyer.Modular_A.Safety.LightCurtain_Stamping := "7A_LIGHT_CURTAIN_1";
	    END_REGION
	    
	    REGION Door
	        "DEV_7".Convoyer.Modular_A.Safety.DoorFront := "7A_DOOR_1";
	        "DEV_7".Convoyer.Modular_A.Safety.DoorBack := "7A_DOOR_2";
	        "DEV_7".Convoyer.Modular_A.Safety.DoorUnload := "7A_DOOR_3";
	    END_REGION
	    
	    REGION Camera
	      //  "DEV".Convoyer_7.Modular_7A.CameraConnection := "MainPLC_Connection_DB";
	    END_REGION
	END_REGION
	REGION 7B
	    REGION Button box left
	        "DEV_7".Convoyer.Modular_B.ButtonControl.ButtonBoxLeft.ButtonReset := "7B_BUTTON_RESET_1";
	        "DEV_7".Convoyer.Modular_B.ButtonControl.ButtonBoxLeft.ButtonStart := "7B_BUTTON_START_1";
	        "DEV_7".Convoyer.Modular_B.ButtonControl.ButtonBoxLeft.ButtonStop := "7B_BUTTON_STOP_1";
	        "DEV_7".Convoyer.Modular_B.Safety.ESTOP_Left := "7B_ESTOP_1";
	    END_REGION
	    
	    REGION Button box right
	        "DEV_7".Convoyer.Modular_B.ButtonControl.ButtonBoxRight.ButtonReset := "7B_BUTTON_RESET_2";
	        "DEV_7".Convoyer.Modular_B.ButtonControl.ButtonBoxRight.ButtonStart := "7B_BUTTON_START_2";
	        "DEV_7".Convoyer.Modular_B.ButtonControl.ButtonBoxRight.ButtonStop := "7B_BUTTON_STOP_2";
	        "DEV_7".Convoyer.Modular_B.Safety.ESTOP_Right := "7B_ESTOP_2";
	    END_REGION
	    
	    REGION Main Cabinet    
	        "DEV_7".Convoyer.Modular_B.ButtonControl.CabinetBox.ButtonReset := "7_BUTTON_RESET";
	        "DEV_7".Convoyer.Modular_B.Safety.ESTOP_MAIN := "7_ESTOP";
	    END_REGION
	    
	    REGION Pneumatics
	        "DEV_7".Convoyer.Modular_B.Pneumatics.Stamping.Sensors.In := "7B_ActuatorIn";
	        "DEV_7".Convoyer.Modular_B.Pneumatics.Stamping.Sensors.Out := "7B_ActuatorOut";
	        "DEV_7".Convoyer.Modular_B.Pneumatics.IVT.Sensor.Analog.RealValue := "7B_IVT_InputSignal_1";
	        "DEV_7".Convoyer.Modular_B.Pneumatics.IVT.Sensor.Scaled.RealNorm := NORM_X(MIN := 0, VALUE := "DEV_7".Convoyer.Modular_B.Pneumatics.IVT.Sensor.Analog.RealValue, MAX := 32767);
	        "DEV_7".Convoyer.Modular_B.Pneumatics.IVT.Sensor.Scaled.RealScale := SCALE_X(MIN := 0, VALUE := "DEV_7".Convoyer.Modular_B.Pneumatics.IVT.Sensor.Scaled.RealNorm, MAX := 7);
	    END_REGION
	    
	    REGION Sensors
	        "DEV_7".Convoyer.Modular_B.Sensors.Homing_I := "7B_Homing_I";
	        "DEV_7".Convoyer.Modular_B.Sensors.Homing_R := "7B_Homing_R";
	        "DEV_7".Convoyer.Modular_B.Sensors.StampingPresence := "7B_StampingPresence" AND "DEV_7".Convoyer.Modular_B.HMI.Stamping.Enable;
	        "DEV_7".Convoyer.Modular_B.Sensors.Stamp_Check_1 := "7B_StampingCheck_1";
	        "DEV_7".Convoyer.Modular_B.Sensors.Stamp_Check_2 := "7B_StampingCheck_2";
	        "DEV_7".Convoyer.Modular_B.Sensors.BlowPresence := NOT "7B_BlowPresence";
	        "DEV_7".Convoyer.Modular_B.Sensors.CameraPresence := "7B_CameraPresence";
	        "DEV_7".Convoyer.Modular_B.Sensors.UnloadingPresence := "7B_UnloadingPresence";
	        "DEV_7".Convoyer.Modular_B.Sensors.Span := "7B_Span";
	        "DEV_7".Convoyer.Modular_B.Sensors.JogBack := "7B_JogBack";
	    END_REGION
	    
	    REGION Light curtains
	        "DEV_7".Convoyer.Modular_B.Safety.LightCurtain_Stamping := "7B_LIGHT_CURTAIN_1";
	    END_REGION
	    
	    REGION Door
	        "DEV_7".Convoyer.Modular_B.Safety.DoorFront := "7B_DOOR_1";
	        "DEV_7".Convoyer.Modular_B.Safety.DoorBack := "7B_DOOR_2";
	        "DEV_7".Convoyer.Modular_B.Safety.DoorUnload := "7B_DOOR_3";
	    END_REGION
	END_REGION
	
	REGION 10A
	    REGION Button box left
	        "DEV_10".Convoyer.Modular_A.ButtonControl.ButtonBoxLeft.ButtonReset := "10A_BUTTON_RESET_1";
	        "DEV_10".Convoyer.Modular_A.ButtonControl.ButtonBoxLeft.ButtonStart := "10A_BUTTON_START_1";
	        "DEV_10".Convoyer.Modular_A.ButtonControl.ButtonBoxLeft.ButtonStop := "10A_BUTTON_STOP_1";
	        "DEV_10".Convoyer.Modular_A.Safety.ESTOP_Left := "10A_ESTOP_1";
	    END_REGION
	    REGION Button box right
	        "DEV_10".Convoyer.Modular_A.ButtonControl.ButtonBoxRight.ButtonReset := "10A_BUTTON_RESET_2";
	        "DEV_10".Convoyer.Modular_A.ButtonControl.ButtonBoxRight.ButtonStart := "10A_BUTTON_START_2";
	        "DEV_10".Convoyer.Modular_A.ButtonControl.ButtonBoxRight.ButtonStop := "10A_BUTTON_STOP_2";
	        "DEV_10".Convoyer.Modular_A.Safety.ESTOP_Right := "10A_ESTOP_2";
	    END_REGION
	    REGION Main Cabinet    
	        "DEV_10".Convoyer.Modular_A.ButtonControl.CabinetBox.ButtonReset := "10_BUTTON_RESET";
	        "DEV_10".Convoyer.Modular_A.Safety.ESTOP_MAIN := "10_ESTOP";
	    END_REGION
	    REGION Pneumatics
	        "DEV_10".Convoyer.Modular_A.Pneumatics.Stamping.Sensors.In := "10A_ActuatorIn";
	        "DEV_10".Convoyer.Modular_A.Pneumatics.Stamping.Sensors.Out := "10A_ActuatorOut";
	        "DEV_10".Convoyer.Modular_A.Pneumatics.IVT.Sensor.Analog.RealValue := "10A_IVT_InputSignal_1";
	        "DEV_10".Convoyer.Modular_A.Pneumatics.IVT.Sensor.Scaled.RealNorm := NORM_X(MIN := 0, VALUE := "DEV_10".Convoyer.Modular_A.Pneumatics.IVT.Sensor.Analog.RealValue, MAX := 32767);
	        "DEV_10".Convoyer.Modular_A.Pneumatics.IVT.Sensor.Scaled.RealScale := SCALE_X(MIN := 0, VALUE := "DEV_10".Convoyer.Modular_A.Pneumatics.IVT.Sensor.Scaled.RealNorm, MAX := 7);
	    END_REGION
	    
	    REGION Sensors
	        "DEV_10".Convoyer.Modular_A.Sensors.Homing_I := "10A_Homing_I";
	        "DEV_10".Convoyer.Modular_A.Sensors.Homing_R := "10A_Homing_R";
	        "DEV_10".Convoyer.Modular_A.Sensors.StampingPresence := "10A_StampingPresence" AND "DEV_10".Convoyer.Modular_A.HMI.Stamping.Enable;
	        "DEV_10".Convoyer.Modular_A.Sensors.Stamp_Check_1 := "10A_StampingCheck_1";
	        "DEV_10".Convoyer.Modular_A.Sensors.Stamp_Check_2 := "10A_StampingCheck_2";
	        "DEV_10".Convoyer.Modular_A.Sensors.BlowPresence := "10A_BlowPresence";
	        "DEV_10".Convoyer.Modular_A.Sensors.CameraPresence := "10A_CameraPresence";
	        "DEV_10".Convoyer.Modular_A.Sensors.UnloadingPresence := "10A_UnloadingPresence";
	        "DEV_10".Convoyer.Modular_A.Sensors.Span := "10A_Span";
	        "DEV_10".Convoyer.Modular_A.Sensors.JogBack := "10A_JogBack";
	    END_REGION
	    
	    REGION Light curtains
	        "DEV_10".Convoyer.Modular_A.Safety.LightCurtain_Stamping := "10A_LIGHT_CURTAIN_1";
	    END_REGION
	    
	    REGION Door
	        "DEV_10".Convoyer.Modular_A.Safety.DoorFront := "10A_DOOR_1";
	        "DEV_10".Convoyer.Modular_A.Safety.DoorBack := "10A_DOOR_2";
	        "DEV_10".Convoyer.Modular_A.Safety.DoorUnload := "10A_DOOR_3";
	    END_REGION
	    
	    REGION Camera
	        //  "DEV".Convoyer_7.Modular_7A.CameraConnection := "MainPLC_Connection_DB";
	    END_REGION
	END_REGION
	
	REGION Thermostat
	    "DEV_7".Convoyer.Modular_A.Safety.Thermostat := NOT "7_THERMOSTAT";
	    "DEV_7".Convoyer.Modular_B.Safety.Thermostat := NOT "7_THERMOSTAT";
	    "DEV_10".Convoyer.Modular_A.Safety.Thermostat := NOT "10_THERMOSTAT";
	END_REGION
	
	REGION 24 v
	    "DEV_7".Convoyer.Diagnostic.Fault_24V := NOT "7_24V_OK";
	    //ZMIENIC PO TESTACH
	    "DEV_10".Convoyer.Diagnostic.Fault_24V := FALSE;
	END_REGION
	
	REGION HMI RECIPE
	    REGION 7A
	        IF "DEV_7".Recipes.Convoyer.A.Type = 0 THEN
	            "DEV_7".Convoyer.Modular_A.HMI.Stamping := "DEV_7".Recipes.Convoyer.A.StampingPL;
	            "DEV_7".Convoyer.Modular_A.HMI.Camera.Enable := "DEV_7".Recipes.Convoyer.A.SettingsPL.Camera;
	            "DEV_7".Convoyer.Modular_A.HMI.Blow.Enable := "DEV_7".Recipes.Convoyer.A.SettingsPL.Blow;
	            "DEV_7".Convoyer.Modular_A.HMI.Blow."Time" := "DEV_7".Recipes.Convoyer.A.SettingsPL.BlowTime;
	        ELSIF "DEV_7".Recipes.Convoyer.A.Type = 1 THEN
	            "DEV_7".Convoyer.Modular_A.HMI.Stamping := "DEV_7".Recipes.Convoyer.A.StampingCN;
	            "DEV_7".Convoyer.Modular_A.HMI.Camera.Enable := "DEV_7".Recipes.Convoyer.A.SettingsCN.Camera;
	            "DEV_7".Convoyer.Modular_A.HMI.Blow.Enable := "DEV_7".Recipes.Convoyer.A.SettingsCN.Blow;
	            "DEV_7".Convoyer.Modular_A.HMI.Blow."Time" := "DEV_7".Recipes.Convoyer.A.SettingsCN.BlowTime;
	        ELSIF "DEV_7".Recipes.Convoyer.A.Type = 2 THEN
	            "DEV_7".Convoyer.Modular_A.HMI.Stamping := "DEV_7".Recipes.Convoyer.A.StampingPlastic;
	            "DEV_7".Convoyer.Modular_A.HMI.Camera.Enable := "DEV_7".Recipes.Convoyer.A.SettingsPlastic.Camera;
	            "DEV_7".Convoyer.Modular_A.HMI.Blow.Enable := "DEV_7".Recipes.Convoyer.A.SettingsPlastic.Blow;
	            "DEV_7".Convoyer.Modular_A.HMI.Blow."Time" := "DEV_7".Recipes.Convoyer.A.SettingsPlastic.BlowTime;
	        ELSIF "DEV_7".Recipes.Convoyer.A.Type = 3 THEN
	            "DEV_7".Convoyer.Modular_A.HMI.Stamping := "DEV_7".Recipes.Convoyer.A.StampingTransport;
	            "DEV_7".Convoyer.Modular_A.HMI.Camera.Enable := "DEV_7".Recipes.Convoyer.A.SettingsTransport.Camera;
	            "DEV_7".Convoyer.Modular_A.HMI.Blow.Enable := "DEV_7".Recipes.Convoyer.A.SettingsTransport.Blow;
	            "DEV_7".Convoyer.Modular_A.HMI.Blow."Time" := "DEV_7".Recipes.Convoyer.A.SettingsTransport.BlowTime;
	        END_IF;
	    END_REGION
	    
	    REGION 7B
	        IF "DEV_7".Recipes.Convoyer.B.Type = 0 THEN
	            "DEV_7".Convoyer.Modular_B.HMI.Stamping := "DEV_7".Recipes.Convoyer.B.StampingPL;
	            "DEV_7".Convoyer.Modular_B.HMI.Camera.Enable := "DEV_7".Recipes.Convoyer.B.SettingsPL.Camera;
	            "DEV_7".Convoyer.Modular_B.HMI.Blow.Enable := "DEV_7".Recipes.Convoyer.B.SettingsPL.Blow;
	            "DEV_7".Convoyer.Modular_B.HMI.Blow."Time" := "DEV_7".Recipes.Convoyer.B.SettingsPL.BlowTime;
	        ELSIF "DEV_7".Recipes.Convoyer.B.Type = 1 THEN
	            "DEV_7".Convoyer.Modular_B.HMI.Stamping := "DEV_7".Recipes.Convoyer.B.StampingCN;
	            "DEV_7".Convoyer.Modular_B.HMI.Camera.Enable := "DEV_7".Recipes.Convoyer.B.SettingsCN.Camera;
	            "DEV_7".Convoyer.Modular_B.HMI.Blow.Enable := "DEV_7".Recipes.Convoyer.B.SettingsCN.Blow;
	            "DEV_7".Convoyer.Modular_B.HMI.Blow."Time" := "DEV_7".Recipes.Convoyer.B.SettingsCN.BlowTime;
	        ELSIF "DEV_7".Recipes.Convoyer.B.Type = 2 THEN
	            "DEV_7".Convoyer.Modular_B.HMI.Stamping := "DEV_7".Recipes.Convoyer.B.StampingPlastic;
	            "DEV_7".Convoyer.Modular_B.HMI.Camera.Enable := "DEV_7".Recipes.Convoyer.B.SettingsPlastic.Camera;
	            "DEV_7".Convoyer.Modular_B.HMI.Blow.Enable := "DEV_7".Recipes.Convoyer.B.SettingsPlastic.Blow;
	            "DEV_7".Convoyer.Modular_B.HMI.Blow."Time" := "DEV_7".Recipes.Convoyer.B.SettingsPlastic.BlowTime;
	        ELSIF "DEV_7".Recipes.Convoyer.B.Type = 3 THEN
	            "DEV_7".Convoyer.Modular_B.HMI.Stamping := "DEV_7".Recipes.Convoyer.B.StampingTransport;
	            "DEV_7".Convoyer.Modular_B.HMI.Camera.Enable := "DEV_7".Recipes.Convoyer.B.SettingsTransport.Camera;
	            "DEV_7".Convoyer.Modular_B.HMI.Blow.Enable := "DEV_7".Recipes.Convoyer.B.SettingsTransport.Blow;
	            "DEV_7".Convoyer.Modular_B.HMI.Blow."Time" := "DEV_7".Recipes.Convoyer.B.SettingsTransport.BlowTime;
	        END_IF;
	    END_REGION
	    
	    REGION 10A
	        IF "DEV_10".Recipes.Convoyer.A.Type = 0 THEN
	            "DEV_10".Convoyer.Modular_A.HMI.Stamping := "DEV_10".Recipes.Convoyer.A.StampingPL;
	            "DEV_10".Convoyer.Modular_A.HMI.Camera.Enable := "DEV_10".Recipes.Convoyer.A.SettingsPL.Camera;
	            "DEV_10".Convoyer.Modular_A.HMI.Blow.Enable := "DEV_10".Recipes.Convoyer.A.SettingsPL.Blow;
	            "DEV_10".Convoyer.Modular_A.HMI.Blow."Time" := "DEV_10".Recipes.Convoyer.A.SettingsPL.BlowTime;
	        ELSIF "DEV_10".Recipes.Convoyer.A.Type = 1 THEN
	            "DEV_10".Convoyer.Modular_A.HMI.Stamping := "DEV_10".Recipes.Convoyer.A.StampingCN;
	            "DEV_10".Convoyer.Modular_A.HMI.Camera.Enable := "DEV_10".Recipes.Convoyer.A.SettingsCN.Camera;
	            "DEV_10".Convoyer.Modular_A.HMI.Blow.Enable := "DEV_10".Recipes.Convoyer.A.SettingsCN.Blow;
	            "DEV_10".Convoyer.Modular_A.HMI.Blow."Time" := "DEV_10".Recipes.Convoyer.A.SettingsCN.BlowTime;
	        ELSIF "DEV_10".Recipes.Convoyer.A.Type = 2 THEN
	            "DEV_10".Convoyer.Modular_A.HMI.Stamping := "DEV_10".Recipes.Convoyer.A.StampingPlastic;
	            "DEV_10".Convoyer.Modular_A.HMI.Camera.Enable := "DEV_10".Recipes.Convoyer.A.SettingsPlastic.Camera;
	            "DEV_10".Convoyer.Modular_A.HMI.Blow.Enable := "DEV_10".Recipes.Convoyer.A.SettingsPlastic.Blow;
	            "DEV_10".Convoyer.Modular_A.HMI.Blow."Time" := "DEV_10".Recipes.Convoyer.A.SettingsPlastic.BlowTime;
	        ELSIF "DEV_10".Recipes.Convoyer.A.Type = 3 THEN
	            "DEV_10".Convoyer.Modular_A.HMI.Stamping := "DEV_10".Recipes.Convoyer.A.StampingTransport;
	            "DEV_10".Convoyer.Modular_A.HMI.Camera.Enable := "DEV_10".Recipes.Convoyer.A.SettingsTransport.Camera;
	            "DEV_10".Convoyer.Modular_A.HMI.Blow.Enable := "DEV_10".Recipes.Convoyer.A.SettingsTransport.Blow;
	            "DEV_10".Convoyer.Modular_A.HMI.Blow."Time" := "DEV_10".Recipes.Convoyer.A.SettingsTransport.BlowTime;
	        END_IF;
	    END_REGION
	END_REGION
	
	
END_FUNCTION

FUNCTION "FC_003_Alarms" : Void
{ S7_Optimized_Access := 'TRUE' }
VERSION : 0.1
   VAR_INPUT 
      StatusInverter_7A : "Status";
      StatusCamera_7A : "Status";
      StatusStamping_7A : "Status";
      StatusInverter_7B : "Status";
      StatusCamera_7B : "Status";
      StatusStamping_7B : "Status";
      StatusInverter_10A : "Status";
      StatusCamera_10A : "Status";
      StatusStamping_10A : "Status";
      Diagnostic_7 : "DiagnosticMainCabinet";
      Diagnostic_10 : "DiagnosticMainCabinet";
   END_VAR

   VAR_IN_OUT 
      Alarms_7A : "Alarms_10";
      Alarms_7B : "Alarms_10";
      Alarms_10A : "Alarms_10";
   END_VAR


BEGIN
	//************************************************************
	//===Author: Mateusz Połojko
	//-----Linkedin: https://pl.linkedin.com/in/mateusz-po%C5%82ojko-52a3541b1
	//-----Github: https://github.com/Bhazel95
	//===Description:
	//-----Alarm triggers
	//===Customer:
	//-----Apator Powogaz S.A.
	//************************************************************
	
	REGION Alarms Convoyer 7
	    #Alarms_7A.ESTOP.Main :=NOT "7_ESTOP";
	    #Alarms_7A.Fault24V := NOT "7_24V_OK";
	    REGION Convoyer 7A   
	        #Alarms_7A.ResetReq := "DEV_7".Convoyer.Modular_A.Safety.REQ_RESET OR NOT "7A_Valve_Safety_1";
	        
	        REGION ESTOP&DOOR
	            #Alarms_7A.ESTOP.Left := NOT "7A_ESTOP_1";
	            #Alarms_7A.ESTOP.Right := NOT "7A_ESTOP_2";
	            #Alarms_7A.Door.Front := NOT "7A_DOOR_1" AND NOT "DEV_7".Convoyer.Modular_A.HMI.DoorDisable.FrontDoor;
	            #Alarms_7A.Door.Back := NOT "7A_DOOR_2" AND NOT "DEV_7".Convoyer.Modular_A.HMI.DoorDisable.BackDoor;
	            #Alarms_7A.Door.Unload := NOT "7A_DOOR_3" AND NOT "DEV_7".Convoyer.Modular_A.HMI.DoorDisable.UnloadDoor;
	        END_REGION
	        REGION Light curtain
	            #Alarms_7A.LightCurtain.Front := (("DEV_7".Convoyer.Modular_A.Pneumatics.Stamping.Coils.In OR "DEV_7".Convoyer.Modular_A.Pneumatics.Stamping.Coils.Out) AND NOT "7A_LIGHT_CURTAIN_1") OR (NOT "DEV_7".Convoyer.Modular_A.Safety.SafetyOK AND NOT "7A_LIGHT_CURTAIN_1");
	        END_REGION
	        
	        REGION INVERTER
	            IF NOT "DEV_7".Convoyer.Modular_A.Safety.REQ_RESET AND "DEV_7".Convoyer.Modular_A.Safety.SafetyOK THEN
	                #Alarms_7A.Inverter.GlobalError := NOT "DEV_7".Convoyer.Modular_A.Safety.InverterOK;
	                #Alarms_7A.Inverter.POWER := #StatusInverter_7A.Error AND #StatusInverter_7A.ErrorStatus = 16#8002;
	                #Alarms_7A.Inverter.HALT := #StatusInverter_7A.Error AND #StatusInverter_7A.ErrorStatus = 16#8001;
	                #Alarms_7A.Inverter.RESET := #StatusInverter_7A.Error AND #StatusInverter_7A.ErrorStatus = 16#8005;
	                #Alarms_7A.Inverter.JOG := #StatusInverter_7A.Error AND #StatusInverter_7A.ErrorStatus = 16#8003;
	                #Alarms_7A.Inverter.RELATIVE := #StatusInverter_7A.Error AND #StatusInverter_7A.ErrorStatus = 16#8004;
	                #Alarms_7A.Inverter.HOMING := #StatusInverter_7A.Error AND #StatusInverter_7A.ErrorStatus = 16#8000;
	            END_IF;
	        END_REGION
	        
	        REGION Camera
	            #Alarms_7A.Camera.ConnectionTimeout := #StatusCamera_7A.Error AND #StatusCamera_7A.ErrorStatus = 16#8000;
	            #Alarms_7A.Camera.MachienStartWrongResponse := #StatusCamera_7A.Error AND #StatusCamera_7A.ErrorStatus = 16#8001;
	            #Alarms_7A.Camera.MachineStartNotSend := #StatusCamera_7A.Error AND #StatusCamera_7A.ErrorStatus = 16#8002;
	            #Alarms_7A.Camera.MachineStartNoResponse := #StatusCamera_7A.Error AND #StatusCamera_7A.ErrorStatus = 16#8003;
	            #Alarms_7A.Camera.CameraWrongResponse := #StatusCamera_7A.Error AND #StatusCamera_7A.ErrorStatus = 16#8004;
	            #Alarms_7A.Camera.CameraNoResponse := #StatusCamera_7A.Error AND #StatusCamera_7A.ErrorStatus = 16#8005;
	            #Alarms_7A.Camera.CameraNotSend := #StatusCamera_7A.Error AND #StatusCamera_7A.ErrorStatus = 16#8006;
	            #Alarms_7A.Camera.TRCV := #StatusCamera_7A.Error AND #StatusCamera_7A.ErrorStatus = 16#8007;
	            #Alarms_7A.Camera.WatchdogTRCV := #StatusCamera_7A.Error AND #StatusCamera_7A.ErrorStatus = 16#8008;
	            #Alarms_7A.Camera.TCON := #StatusCamera_7A.Error AND #StatusCamera_7A.ErrorStatus = 16#8009;
	            #Alarms_7A.Camera.TDISCON := #StatusCamera_7A.Error AND #StatusCamera_7A.ErrorStatus = 16#8010;
	            #Alarms_7A.Camera.TSEND := #StatusCamera_7A.Error AND #StatusCamera_7A.ErrorStatus = 16#8011;
	        END_REGION
	        
	        REGION "Stamping"
	            #Alarms_7A.Pneumatics.Span := NOT "7A_Span";
	            #Alarms_7A.Pneumatics.Stamping.NotHomed := #StatusStamping_7A.Error AND #StatusStamping_7A.ErrorStatus = 16#8000;
	            #Alarms_7A.Pneumatics.Stamping.WatchdogIn := #StatusStamping_7A.Error AND #StatusStamping_7A.ErrorStatus = 16#8001;
	            #Alarms_7A.Pneumatics.Stamping.WatchdogOut := #StatusStamping_7A.Error AND #StatusStamping_7A.ErrorStatus = 16#8002;
	        END_REGION
	        
	        REGION IVT
	            ;
	        END_REGION
	    END_REGION
	    END_REGION
	    
	    REGION Convoyer 7B 
	        #Alarms_7B.ResetReq := "DEV_7".Convoyer.Modular_B.Safety.REQ_RESET OR NOT "7B_Valve_Safety_1";
	        REGION ESTOP&DOOR
	            #Alarms_7B.ESTOP.Left := NOT "7B_ESTOP_1";
	            #Alarms_7B.ESTOP.Right := NOT "7B_ESTOP_2";
	            #Alarms_7B.Door.Front := NOT "7B_DOOR_1" AND NOT "DEV_7".Convoyer.Modular_B.HMI.DoorDisable.FrontDoor;
	            #Alarms_7B.Door.Back := NOT "7B_DOOR_2" AND NOT "DEV_7".Convoyer.Modular_B.HMI.DoorDisable.BackDoor;
	            #Alarms_7B.Door.Unload := NOT "7B_DOOR_3" AND NOT "DEV_7".Convoyer.Modular_B.HMI.DoorDisable.UnloadDoor;
	        END_REGION
	        REGION Light curtain
	            #Alarms_7B.LightCurtain.Front := (("DEV_7".Convoyer.Modular_B.Pneumatics.Stamping.Coils.In OR "DEV_7".Convoyer.Modular_B.Pneumatics.Stamping.Coils.Out) AND NOT "7B_LIGHT_CURTAIN_1") OR (NOT "DEV_7".Convoyer.Modular_B.Safety.SafetyOK AND NOT "7B_LIGHT_CURTAIN_1");
	        END_REGION
	        
	        REGION INVERTER
	            IF NOT "DEV_7".Convoyer.Modular_B.Safety.REQ_RESET AND "DEV_7".Convoyer.Modular_B.Safety.SafetyOK THEN
	                #Alarms_7B.Inverter.GlobalError := NOT "DEV_7".Convoyer.Modular_B.Safety.InverterOK;
	                #Alarms_7B.Inverter.POWER := #StatusInverter_7B.Error AND #StatusInverter_7B.ErrorStatus = 16#8002;
	                #Alarms_7B.Inverter.HALT := #StatusInverter_7B.Error AND #StatusInverter_7B.ErrorStatus = 16#8001;
	                #Alarms_7B.Inverter.RESET := #StatusInverter_7B.Error AND #StatusInverter_7B.ErrorStatus = 16#8005;
	                #Alarms_7B.Inverter.JOG := #StatusInverter_7B.Error AND #StatusInverter_7B.ErrorStatus = 16#8003;
	                #Alarms_7B.Inverter.RELATIVE := #StatusInverter_7B.Error AND #StatusInverter_7B.ErrorStatus = 16#8004;
	                #Alarms_7B.Inverter.HOMING := #StatusInverter_7B.Error AND #StatusInverter_7B.ErrorStatus = 16#8000;
	            END_IF;
	        END_REGION
	        
	        REGION Camera
	            #Alarms_7B.Camera.ConnectionTimeout := #StatusCamera_7B.Error AND #StatusCamera_7B.ErrorStatus = 16#8000;
	            #Alarms_7B.Camera.MachienStartWrongResponse := #StatusCamera_7B.Error AND #StatusCamera_7B.ErrorStatus = 16#8001;
	            #Alarms_7B.Camera.MachineStartNotSend := #StatusCamera_7B.Error AND #StatusCamera_7B.ErrorStatus = 16#8002;
	            #Alarms_7B.Camera.MachineStartNoResponse := #StatusCamera_7B.Error AND #StatusCamera_7B.ErrorStatus = 16#8003;
	            #Alarms_7B.Camera.CameraWrongResponse := #StatusCamera_7B.Error AND #StatusCamera_7B.ErrorStatus = 16#8004;
	            #Alarms_7B.Camera.CameraNoResponse := #StatusCamera_7B.Error AND #StatusCamera_7B.ErrorStatus = 16#8005;
	            #Alarms_7B.Camera.CameraNotSend := #StatusCamera_7B.Error AND #StatusCamera_7B.ErrorStatus = 16#8006;
	            #Alarms_7B.Camera.TRCV := #StatusCamera_7B.Error AND #StatusCamera_7B.ErrorStatus = 16#8007;
	            #Alarms_7B.Camera.WatchdogTRCV := #StatusCamera_7B.Error AND #StatusCamera_7B.ErrorStatus = 16#8008;
	            #Alarms_7B.Camera.TCON := #StatusCamera_7B.Error AND #StatusCamera_7B.ErrorStatus = 16#8009;
	            #Alarms_7B.Camera.TDISCON := #StatusCamera_7B.Error AND #StatusCamera_7B.ErrorStatus = 16#8010;
	            #Alarms_7B.Camera.TSEND := #StatusCamera_7B.Error AND #StatusCamera_7B.ErrorStatus = 16#8011;
	        END_REGION
	        
	        REGION "Stamping"
	            #Alarms_7B.Pneumatics.Span := NOT "7B_Span";
	            #Alarms_7B.Pneumatics.Stamping.NotHomed := #StatusStamping_7B.Error AND #StatusStamping_7B.ErrorStatus = 16#8000;
	            #Alarms_7B.Pneumatics.Stamping.WatchdogIn := #StatusStamping_7B.Error AND #StatusStamping_7B.ErrorStatus = 16#8001;
	            #Alarms_7B.Pneumatics.Stamping.WatchdogOut := #StatusStamping_7B.Error AND #StatusStamping_7B.ErrorStatus = 16#8002;
	        END_REGION
	        
	        REGION IVT
	            ;
	        END_REGION
	    END_REGION 
	    
	    
	    REGION Alarms Convoyer 10
	        #Alarms_10A.ESTOP.Main := NOT "10_ESTOP";
	        //do zmiany
	        #Alarms_10A.Fault24V := FALSE;
	        REGION Convoyer 10A   
	            #Alarms_10A.ResetReq := "DEV_10".Convoyer.Modular_A.Safety.REQ_RESET OR NOT "10A_Valve_Safety_1";
	            
	            REGION ESTOP&DOOR
	                #Alarms_10A.ESTOP.Left := NOT "10A_ESTOP_1";
	                #Alarms_10A.ESTOP.Right := NOT "10A_ESTOP_2";
	                #Alarms_10A.Door.Front := NOT "10A_DOOR_1" AND NOT "DEV_10".Convoyer.Modular_A.HMI.DoorDisable.FrontDoor;
	                #Alarms_10A.Door.Back := NOT "10A_DOOR_2" AND NOT "DEV_10".Convoyer.Modular_A.HMI.DoorDisable.BackDoor;
	                #Alarms_10A.Door.Unload := NOT "10A_DOOR_3" AND NOT "DEV_10".Convoyer.Modular_A.HMI.DoorDisable.UnloadDoor;
	            END_REGION
	            REGION Light curtain
	                #Alarms_10A.LightCurtain.Front := (("DEV_10".Convoyer.Modular_A.Pneumatics.Stamping.Coils.In OR "DEV_10".Convoyer.Modular_A.Pneumatics.Stamping.Coils.Out) AND NOT "10A_LIGHT_CURTAIN_1") OR (NOT "DEV_10".Convoyer.Modular_A.Safety.SafetyOK AND NOT "10A_LIGHT_CURTAIN_1");
	            END_REGION
	            
	            REGION INVERTER
	                IF NOT "DEV_10".Convoyer.Modular_A.Safety.REQ_RESET AND "DEV_10".Convoyer.Modular_A.Safety.SafetyOK THEN
	                    #Alarms_10A.Inverter.GlobalError := NOT "DEV_10".Convoyer.Modular_A.Safety.InverterOK;
	                    #Alarms_10A.Inverter.POWER := #StatusInverter_10A.Error AND #StatusInverter_10A.ErrorStatus = 16#8002;
	                    #Alarms_10A.Inverter.HALT := #StatusInverter_10A.Error AND #StatusInverter_10A.ErrorStatus = 16#8001;
	                    #Alarms_10A.Inverter.RESET := #StatusInverter_10A.Error AND #StatusInverter_10A.ErrorStatus = 16#8005;
	                    #Alarms_10A.Inverter.JOG := #StatusInverter_10A.Error AND #StatusInverter_10A.ErrorStatus = 16#8003;
	                    #Alarms_10A.Inverter.RELATIVE := #StatusInverter_10A.Error AND #StatusInverter_10A.ErrorStatus = 16#8004;
	                    #Alarms_10A.Inverter.HOMING := #StatusInverter_10A.Error AND #StatusInverter_10A.ErrorStatus = 16#8000;
	                END_IF;
	            END_REGION
	            
	            REGION Camera
	                #Alarms_10A.Camera.ConnectionTimeout := #StatusCamera_10A.Error AND #StatusCamera_10A.ErrorStatus = 16#8000;
	                #Alarms_10A.Camera.MachienStartWrongResponse := #StatusCamera_10A.Error AND #StatusCamera_10A.ErrorStatus = 16#8001;
	                #Alarms_10A.Camera.MachineStartNotSend := #StatusCamera_10A.Error AND #StatusCamera_10A.ErrorStatus = 16#8002;
	                #Alarms_10A.Camera.MachineStartNoResponse := #StatusCamera_10A.Error AND #StatusCamera_10A.ErrorStatus = 16#8003;
	                #Alarms_10A.Camera.CameraWrongResponse := #StatusCamera_10A.Error AND #StatusCamera_10A.ErrorStatus = 16#8004;
	                #Alarms_10A.Camera.CameraNoResponse := #StatusCamera_10A.Error AND #StatusCamera_10A.ErrorStatus = 16#8005;
	                #Alarms_10A.Camera.CameraNotSend := #StatusCamera_10A.Error AND #StatusCamera_10A.ErrorStatus = 16#8006;
	                #Alarms_10A.Camera.TRCV := #StatusCamera_10A.Error AND #StatusCamera_10A.ErrorStatus = 16#8007;
	                #Alarms_10A.Camera.WatchdogTRCV := #StatusCamera_10A.Error AND #StatusCamera_10A.ErrorStatus = 16#8008;
	                #Alarms_10A.Camera.TCON := #StatusCamera_10A.Error AND #StatusCamera_10A.ErrorStatus = 16#8009;
	                #Alarms_10A.Camera.TDISCON := #StatusCamera_10A.Error AND #StatusCamera_10A.ErrorStatus = 16#8010;
	                #Alarms_10A.Camera.TSEND := #StatusCamera_10A.Error AND #StatusCamera_10A.ErrorStatus = 16#8011;
	            END_REGION
	            
	            REGION "Stamping"
	                #Alarms_10A.Pneumatics.Span := NOT "10A_Span";
	                #Alarms_10A.Pneumatics.Stamping.NotHomed := #StatusStamping_10A.Error AND #StatusStamping_10A.ErrorStatus = 16#8000;
	                #Alarms_10A.Pneumatics.Stamping.WatchdogIn := #StatusStamping_10A.Error AND #StatusStamping_10A.ErrorStatus = 16#8001;
	                #Alarms_10A.Pneumatics.Stamping.WatchdogOut := #StatusStamping_10A.Error AND #StatusStamping_10A.ErrorStatus = 16#8002;
	            END_REGION
	            
	            REGION IVT
	                ;
	            END_REGION
	        END_REGION
	    END_REGION
	
	    REGION Diagnostic 7
	        #Alarms_7A.Diagnostic.ET200SP.Head := #Diagnostic_7.ET_200SP.HeadModule_0.diagDIS.OwnState <> 0;
	        #Alarms_7A.Diagnostic.ET200SP.BusAdapter := #Diagnostic_7.ET_200SP.BusAdapter_1.diagDIS.OwnState <> 0;
	        #Alarms_7A.Diagnostic.ET200SP.FDI_1 := #Diagnostic_7.ET_200SP.InputSafety_2.diagDIS.OwnState <> 0;
	        #Alarms_7A.Diagnostic.ET200SP.FDI_2 := #Diagnostic_7.ET_200SP.InputSafety_3.diagDIS.OwnState <> 0;
	        #Alarms_7A.Diagnostic.ET200SP.FDI_3 := #Diagnostic_7.ET_200SP.InputSafety_4.diagDIS.OwnState <> 0;
	        #Alarms_7A.Diagnostic.ET200SP.FDI_4 := #Diagnostic_7.ET_200SP.InputSafety_5.diagDIS.OwnState <> 0;
	        #Alarms_7A.Diagnostic.ET200SP.FDI_5 := #Diagnostic_7.ET_200SP.InputSafety_6.diagDIS.OwnState <> 0;
	        #Alarms_7A.Diagnostic.ET200SP.FDQ_1 := #Diagnostic_7.ET_200SP.OutputSafety_7.diagDIS.OwnState <> 0;
	        #Alarms_7A.Diagnostic.ET200SP.FRQ_1 := #Diagnostic_7.ET_200SP.RelaySafety_9.diagDIS.OwnState <> 0;
	        #Alarms_7A.Diagnostic.ET200SP.FRQ_2 := #Diagnostic_7.ET_200SP.RelaySafety_10.diagDIS.OwnState <> 0;
	        #Alarms_7A.Diagnostic.ET200SP.DI_1 := #Diagnostic_7.ET_200SP.InputsDigital_11.diagDIS.OwnState <> 0;
	        #Alarms_7A.Diagnostic.ET200SP.DI_2 := #Diagnostic_7.ET_200SP.InputsDigital_12.diagDIS.OwnState <> 0;
	        #Alarms_7A.Diagnostic.ET200SP.DI_3 := #Diagnostic_7.ET_200SP.InputsDigital_13.diagDIS.OwnState <> 0;
	        #Alarms_7A.Diagnostic.ET200SP.AI_1 := #Diagnostic_7.ET_200SP.InputAnalog_14.diagDIS.OwnState <> 0;
	        #Alarms_7A.Diagnostic.ET200SP.DQ_1 := #Diagnostic_7.ET_200SP.OutputDigital_15.diagDIS.OwnState <> 0;
	        #Alarms_7A.Diagnostic.ET200SP.DQ_2 := #Diagnostic_7.ET_200SP.OutputDigital_16.diagDIS.OwnState <> 0;
	        #Alarms_7A.Diagnostic.ET200SP.DQ_3 := #Diagnostic_7.ET_200SP.OutputDigital_17.diagDIS.OwnState <> 0;
	        #Alarms_7A.Diagnostic.ET200SP.DQ_4 := #Diagnostic_7.ET_200SP.OutputDigital_18.diagDIS.OwnState <> 0;
	        #Alarms_7A.Diagnostic.ET200SP.AQ_1 := #Diagnostic_7.ET_200SP.OutputAnalog_19.diagDIS.OwnState <> 0;
	        #Alarms_7A.Diagnostic.ET200SP.AL_1 := #Diagnostic_7.ET_200SP.ET_200AL_1.diagDIS.OwnState <> 0;
	        #Alarms_7A.Diagnostic.ET200SP.AL_2 := #Diagnostic_7.ET_200SP.ET_200AL_2.diagDIS.OwnState <> 0;
	        #Alarms_7B.Diagnostic.ET200SP.AL_1 := #Diagnostic_7.ET_200SP.ET_200AL_3.diagDIS.OwnState <> 0;
	        #Alarms_7B.Diagnostic.ET200SP.AL_2 := #Diagnostic_7.ET_200SP.ET_200AL_4.diagDIS.OwnState <> 0;
	        
	        #Alarms_7A.Diagnostic.Sinamic_1 := #Diagnostic_7.SinamicG120_1.diagDIS.OwnState <> 0;
	        #Alarms_7B.Diagnostic.Sinamic_1 := #Diagnostic_7.SinamicG120_2.diagDIS.OwnState <> 0;
	        #Alarms_7A.Diagnostic.GeneralDiag := NOT #Diagnostic_7.DiagnosticOK;
	        
	        
	        #Alarms_7A.CriticalALarm := #Alarms_7A.ESTOP.Left OR #Alarms_7A.ESTOP.Right OR #Alarms_7A.ESTOP.Main OR
	        #Alarms_7A.Door.Front OR #Alarms_7A.Door.Back OR #Alarms_7A.Door.Unload;
	        #Alarms_7A.Present := #Alarms_7A.CriticalALarm OR #StatusCamera_7A.Error OR #StatusInverter_7A.Error OR #StatusStamping_7A.Error OR NOT #Diagnostic_7.DiagnosticOK OR #Alarms_7A.Pneumatics.Span;
	        
	        #Alarms_7B.CriticalALarm := #Alarms_7B.ESTOP.Left OR #Alarms_7B.ESTOP.Right OR #Alarms_7B.ESTOP.Main OR
	        #Alarms_7B.Door.Front OR #Alarms_7B.Door.Back OR #Alarms_7B.Door.Unload;
	        #Alarms_7B.Present := #Alarms_7B.CriticalALarm OR #StatusCamera_7B.Error OR #StatusInverter_7B.Error OR #StatusStamping_7B.Error OR NOT #Diagnostic_7.DiagnosticOK OR #Alarms_7B.Pneumatics.Span;
	        
	        
	    END_REGION
	    
	    REGION Diagnostic 10
	        #Alarms_10A.Diagnostic.ET200SP.Head := #Diagnostic_10.ET_200SP.HeadModule_0.diagDIS.OwnState <> 0;
	        #Alarms_10A.Diagnostic.ET200SP.BusAdapter := #Diagnostic_10.ET_200SP.BusAdapter_1.diagDIS.OwnState <> 0;
	        #Alarms_10A.Diagnostic.ET200SP.FDI_1 := #Diagnostic_10.ET_200SP.InputSafety_2.diagDIS.OwnState <> 0;
	        #Alarms_10A.Diagnostic.ET200SP.FDI_2 := #Diagnostic_10.ET_200SP.InputSafety_3.diagDIS.OwnState <> 0;
	        #Alarms_10A.Diagnostic.ET200SP.FDI_3 := #Diagnostic_10.ET_200SP.InputSafety_4.diagDIS.OwnState <> 0;
	        #Alarms_10A.Diagnostic.ET200SP.FDI_4 := #Diagnostic_10.ET_200SP.InputSafety_5.diagDIS.OwnState <> 0;
	        #Alarms_10A.Diagnostic.ET200SP.FDI_5 := #Diagnostic_10.ET_200SP.InputSafety_6.diagDIS.OwnState <> 0;
	        #Alarms_10A.Diagnostic.ET200SP.FDQ_1 := #Diagnostic_10.ET_200SP.OutputSafety_7.diagDIS.OwnState <> 0;
	        #Alarms_10A.Diagnostic.ET200SP.FRQ_1 := #Diagnostic_10.ET_200SP.RelaySafety_9.diagDIS.OwnState <> 0;
	        #Alarms_10A.Diagnostic.ET200SP.FRQ_2 := #Diagnostic_10.ET_200SP.RelaySafety_10.diagDIS.OwnState <> 0;
	        #Alarms_10A.Diagnostic.ET200SP.DI_1 := #Diagnostic_10.ET_200SP.InputsDigital_11.diagDIS.OwnState <> 0;
	        #Alarms_10A.Diagnostic.ET200SP.DI_2 := #Diagnostic_10.ET_200SP.InputsDigital_12.diagDIS.OwnState <> 0;
	        #Alarms_10A.Diagnostic.ET200SP.DI_3 := #Diagnostic_10.ET_200SP.InputsDigital_13.diagDIS.OwnState <> 0;
	        #Alarms_10A.Diagnostic.ET200SP.AI_1 := #Diagnostic_10.ET_200SP.InputAnalog_14.diagDIS.OwnState <> 0;
	        #Alarms_10A.Diagnostic.ET200SP.DQ_1 := #Diagnostic_10.ET_200SP.OutputDigital_15.diagDIS.OwnState <> 0;
	        #Alarms_10A.Diagnostic.ET200SP.DQ_2 := #Diagnostic_10.ET_200SP.OutputDigital_16.diagDIS.OwnState <> 0;
	        #Alarms_10A.Diagnostic.ET200SP.DQ_3 := #Diagnostic_10.ET_200SP.OutputDigital_17.diagDIS.OwnState <> 0;
	        #Alarms_10A.Diagnostic.ET200SP.DQ_4 := #Diagnostic_10.ET_200SP.OutputDigital_18.diagDIS.OwnState <> 0;
	        #Alarms_10A.Diagnostic.ET200SP.AQ_1 := #Diagnostic_10.ET_200SP.OutputAnalog_19.diagDIS.OwnState <> 0;
	        #Alarms_10A.Diagnostic.ET200SP.AL_1 := #Diagnostic_10.ET_200SP.ET_200AL_1.diagDIS.OwnState <> 0;
	        #Alarms_10A.Diagnostic.ET200SP.AL_2 := #Diagnostic_10.ET_200SP.ET_200AL_2.diagDIS.OwnState <> 0;
	        //#Alarms_10B.Diagnostic.ET200SP.AL_1 := #Diagnostic_7.ET_200SP.ET_200AL_3.diagDIS.OwnState <> 0;
	        //#Alarms_10B.Diagnostic.ET200SP.AL_2 := #Diagnostic_7.ET_200SP.ET_200AL_4.diagDIS.OwnState <> 0;
	        
	        #Alarms_10A.Diagnostic.Sinamic_1 := #Diagnostic_10.SinamicG120_1.diagDIS.OwnState <> 0;
	        // #Alarms_7B.Diagnostic.Sinamic_1 := #Diagnostic_7.SinamicG120_2.diagDIS.OwnState <> 0;
	        #Alarms_10A.Diagnostic.GeneralDiag := NOT #Diagnostic_10.DiagnosticOK;
	        
	        
	        #Alarms_10A.CriticalALarm := #Alarms_10A.ESTOP.Left OR #Alarms_10A.ESTOP.Right OR #Alarms_10A.ESTOP.Main OR
	        #Alarms_10A.Door.Front OR #Alarms_10A.Door.Back OR #Alarms_10A.Door.Unload;
	        #Alarms_10A.Present := #Alarms_10A.CriticalALarm OR #StatusCamera_10A.Error OR #StatusInverter_10A.Error OR #StatusStamping_10A.Error OR NOT #Diagnostic_10.DiagnosticOK OR #Alarms_10A.Pneumatics.Span;
	    END_REGION
	
	IF #Alarms_7A.Present THEN
	    "DEV_7".Convoyer.Modular_A.HMI.Page.Number := 1;
	ELSE
	    "DEV_7".Convoyer.Modular_A.HMI.Page.Number := 0;
	END_IF;
	
END_FUNCTION

FUNCTION_BLOCK "Stamping"
{ S7_Optimized_Access := 'TRUE' }
VERSION : 0.1
   VAR_INPUT 
      Reset : Bool;
      SecondPush : Bool;
      TimerSecondPush : Time;
      PreasureSecondPush : Real;
      TimerStamp : Time;
      TimerMax : Time;
      MaxPreasure : Real;
      RegularPreasure : Real;
   END_VAR

   VAR_OUTPUT 
      Status : "Status";
   END_VAR

   VAR_IN_OUT 
      Valve : "Valve5_3";
      ITV : "IVT";
      Execute : Bool;
   END_VAR

   VAR 
      State { S7_SetPoint := 'False'} : "s_changeState";
      Timers : Struct
         SetIn { S7_SetPoint := 'False'} : "s_TON";
         SetOut : "s_TON";
         Stamping : "s_TON";
         SecondPush : "s_TON";
         GoOut : "s_TON";
      END_STRUCT;
      R_TRIG_Exe {InstructionName := 'R_TRIG'; LibVersion := '1.0'; ExternalAccessible := 'False'; ExternalVisible := 'False'; ExternalWritable := 'False'; S7_SetPoint := 'False'} : R_TRIG;
      FirstTry { S7_SetPoint := 'True'} : Bool;
   END_VAR

   VAR CONSTANT 
      S_IDLE : Int := 0;
      S_ERROR : Int := 20;
      S_GO_IN : Int := 30;
      S_GO_OUT : Int := 40;
      NotHomed : Word := 16#8000;
      WatchdogIn : Word := 16#8001;
      WatchdogOut : Word := 16#8002;
   END_VAR


BEGIN
	//************************************************************
	//===Author: Mateusz Połojko
	//-----Linkedin: https://pl.linkedin.com/in/mateusz-po%C5%82ojko-52a3541b1
	//-----Github: https://github.com/Bhazel95
	//===Description:
	//-----Stamping control
	//===Customer:
	//-----Apator Powogaz S.A.
	//************************************************************
	
	REGION #Timers
	    #Timers.SetIn.PT := #Valve.Timers.In;
	    #Timers.SetIn.Timer(IN := #Timers.SetIn.IN,
	                        PT := #Timers.SetIn.PT);
	    
	    #Timers.SetOut.PT := #Valve.Timers.Out;
	    #Timers.SetOut.Timer(IN := #Timers.SetOut.IN,
	                         PT := #Timers.SetOut.PT);
	    
	    #Timers.Stamping.PT := #TimerStamp;
	    #Timers.Stamping.Timer(IN := #Valve.Sensors.Out,
	                           PT := #Timers.Stamping.PT);
	    
	    #Timers.SecondPush.PT := #TimerSecondPush;
	    #Timers.SecondPush.Timer(IN := #Valve.Sensors.Out,
	                             PT := #Timers.SecondPush.PT);
	    
	    #Timers.GoOut.PT := T#300MS;
	    #Timers.GoOut.Timer(IN := #Timers.GoOut.IN,
	                        PT := #Timers.GoOut.PT);
	END_REGION
	#R_TRIG_Exe(CLK:=#Execute);
	
	CASE #State.state OF
	    #S_IDLE:
	        //Funkcja wejścia
	        IF #State.inputFlag AND NOT #State.outputFlag THEN
	            #State.name := 'STAN BEZCZYNNY';
	            #Execute := FALSE;
	            #Status.Busy := FALSE;
	            #Status.Ready := TRUE;
	            #Status.Done := TRUE;
	            #Status.Error := FALSE;
	            #Status.ErrorStatus := 16#0000;
	            #Valve.Coils.In := FALSE;
	            #Valve.Coils.Out := FALSE;
	            #FirstTry := FALSE;
	        END_IF;
	        
	        //Funkcja cykliczna
	        IF NOT #State.inputFlag AND NOT #State.outputFlag THEN
	            #Status.Ready := TRUE;
	            IF #Reset AND NOT #Valve.Sensors.In THEN
	                "changeState"(newState := #S_GO_IN,
	                              Data := #State);
	            END_IF;
	            
	            
	            IF #R_TRIG_Exe.Q THEN
	                IF NOT #Valve.Sensors.In THEN
	                    #Status.ErrorStatus := #NotHomed;
	                    "changeState"(newState := #S_ERROR,
	                                  Data := #State);
	                ELSE
	                    #FirstTry := TRUE;
	                    "changeState"(newState := #S_GO_OUT,
	                                  Data := #State);
	                END_IF;
	            END_IF;
	        END_IF;
	        
	        //Funkcja wyjściowa 
	        IF #State.outputFlag THEN
	            #Status.Done := FALSE;
	        END_IF;
	        
	    #S_ERROR:
	        //Funkcja wejścia
	        IF #State.inputFlag AND NOT #State.outputFlag THEN
	            #State.name := 'ERROR';
	            #Status.Busy := FALSE;
	            #Status.Ready := FALSE;
	            #Status.Done := FALSE;
	            #Status.Error := TRUE;
	            #Valve.Coils.In := FALSE;
	            #Valve.Coils.Out := FALSE;
	            #Timers.GoOut.IN := FALSE;
	            RESET_TIMER(#Timers.GoOut.Timer);
	            #Timers.SecondPush.IN := FALSE;
	            RESET_TIMER(#Timers.SecondPush.Timer);
	            #Timers.SetIn.IN := FALSE;
	            RESET_TIMER(#Timers.SetIn.Timer);
	            #Timers.SetOut.IN:= FALSE;
	            RESET_TIMER(#Timers.SetOut.Timer);
	            #Timers.Stamping.IN := FALSE;
	            RESET_TIMER(#Timers.Stamping.Timer);
	        END_IF;
	        
